LIN {X 70.506,Y 104.962,Z 68.043,A 180.000,B 0.000,C 180.000} C_DIS
LIN {X 70.550,Y 104.810,Z 68.040,A 180.000,B 0.000,C 180.000} C_DIS
LIN {X 70.594,Y 104.659,Z 68.037,A 180.000,B 0.000,C 180.000} C_DIS
LIN {X 70.631,Y 104.506,Z 68.034,A 180.000,B 0.000,C 180.000} C_DIS
LIN {X 70.666,Y 104.352,Z 68.032,A 180.000,B 0.000,C 180.000} C_DIS
LIN {X 70.700,Y 104.199,Z 68.029,A 180.000,B 0.000,C 180.000} C_DIS
LIN {X 70.735,Y 104.045,Z 68.027,A 180.000,B 0.000,C 180.000} C_DIS
LIN {X 70.797,Y 103.736,Z 68.022,A 180.000,B 0.000,C 180.000} C_DIS
LIN {X 70.846,Y 103.425,Z 68.018,A 180.000,B 0.000,C 180.000} C_DIS
LIN {X 70.895,Y 103.114,Z 68.014,A 180.000,B 0.000,C 180.000} C_DIS
LIN {X 70.928,Y 102.801,Z 68.011,A 180.000,B 0.000,C 180.000} C_DIS
LIN {X 70.957,Y 102.487,Z 68.008,A 180.000,B 0.000,C 180.000} C_DIS
LIN {X 70.980,Y 102.173,Z 68.005,A 180.000,B 0.000,C 180.000} C_DIS
LIN {X 70.990,Y 101.858,Z 68.003,A 180.000,B 0.000,C 180.000} C_DIS
LIN {X 71.000,Y 101.543,Z 68.002,A 180.000,B 0.000,C 180.000} C_DIS
LIN {X 70.993,Y 101.228,Z 68.001,A 180.000,B 0.000,C 180.000} C_DIS
LIN {X 70.983,Y 100.914,Z 68.000,A 180.000,B 0.000,C 180.000} C_DIS
LIN {X 70.973,Y 100.682,Z 68.000,A 180.000,B 0.000,C 180.000} C_DIS
; Cutting Move Starts
LIN {X 70.970,Y 100.651,Z 68.000,A 180.000,B 0.000,C 180.000} C_DIS
LIN {X 70.954,Y 100.472,Z 68.000,A 180.000,B 0.000,C 180.000} C_DIS
LIN {X 70.920,Y 100.114,Z 68.000,A 180.000,B 0.000,C 180.000} C_DIS
LIN {X 70.902,Y 99.936,Z 68.000,A 180.000,B 0.000,C 180.000} C_DIS
LIN {X 70.875,Y 99.757,Z 68.000,A 180.000,B 0.000,C 180.000} C_DIS
LIN {X 70.796,Y 99.261,Z 68.000,A 180.000,B 0.000,C 180.000} C_DIS
LIN {X 70.790,Y 99.221,Z 68.000,A 180.000,B 0.000,C 180.000} C_DIS
LIN {X 70.754,Y 99.042,Z 68.000,A 180.000,B 0.000,C 180.000} C_DIS
LIN {X 70.670,Y 98.665,Z 68.000,A 180.000,B 0.000,C 180.000} C_DIS
LIN {X 70.634,Y 98.505,Z 68.000,A 180.000,B 0.000,C 180.000} C_DIS
LIN {X 70.617,Y 98.432,Z 68.000,A 180.000,B 0.000,C 180.000} C_DIS
LIN {X 70.590,Y 98.327,Z 68.000,A 180.000,B 0.000,C 180.000} C_DIS
LIN {X 70.538,Y 98.148,Z 68.000,A 180.000,B 0.000,C 180.000} C_DIS
LIN {X 70.434,Y 97.790,Z 68.000,A 180.000,B 0.000,C 180.000} C_DIS
LIN {X 70.380,Y 97.612,Z 68.000,A 180.000,B 0.000,C 180.000} C_DIS
LIN {X 70.316,Y 97.433,Z 68.000,A 180.000,B 0.000,C 180.000} C_DIS
LIN {X 70.187,Y 97.075,Z 68.000,A 180.000,B 0.000,C 180.000} C_DIS
LIN {X 70.121,Y 96.897,Z 68.000,A 180.000,B 0.000,C 180.000} C_DIS
LIN {X 70.081,Y 96.800,Z 68.000,A 180.000,B 0.000,C 180.000} C_DIS
LIN {X 69.891,Y 96.360,Z 68.000,A 180.000,B 0.000,C 180.000} C_DIS
LIN {X 69.812,Y 96.181,Z 68.000,A 180.000,B 0.000,C 180.000} C_DIS
LIN {X 69.724,Y 96.005,Z 68.000,A 180.000,B 0.000,C 180.000} C_DIS
LIN {X 69.540,Y 95.645,Z 68.000,A 180.000,B 0.000,C 180.000} C_DIS
LIN {X 69.447,Y 95.466,Z 68.000,A 180.000,B 0.000,C 180.000} C_DIS
LIN {X 69.366,Y 95.327,Z 68.000,A 180.000,B 0.000,C 180.000} C_DIS
LIN {X 69.131,Y 94.930,Z 68.000,A 180.000,B 0.000,C 180.000} C_DIS
LIN {X 69.021,Y 94.751,Z 68.000,A 180.000,B 0.000,C 180.000} C_DIS
LIN {X 69.008,Y 94.733,Z 68.000,A 180.000,B 0.000,C 180.000} C_DIS
LIN {X 68.657,Y 94.215,Z 68.000,A 180.000,B 0.000,C 180.000} C_DIS
LIN {X 68.651,Y 94.207,Z 68.000,A 180.000,B 0.000,C 180.000} C_DIS
LIN {X 68.524,Y 94.036,Z 68.000,A 180.000,B 0.000,C 180.000} C_DIS
LIN {X 68.247,Y 93.679,Z 68.000,A 180.000,B 0.000,C 180.000} C_DIS
LIN {X 68.115,Y 93.512,Z 68.000,A 180.000,B 0.000,C 180.000} C_DIS
LIN {X 68.104,Y 93.500,Z 68.000,A 180.000,B 0.000,C 180.000} C_DIS
LIN {X 67.947,Y 93.321,Z 68.000,A 180.000,B 0.000,C 180.000} C_DIS
LIN {X 67.757,Y 93.106,Z 68.000,A 180.000,B 0.000,C 180.000} C_DIS
LIN {X 67.631,Y 92.964,Z 68.000,A 180.000,B 0.000,C 180.000} C_DIS
LIN {X 67.578,Y 92.908,Z 68.000,A 180.000,B 0.000,C 180.000} C_DIS
LIN {X 67.456,Y 92.785,Z 68.000,A 180.000,B 0.000,C 180.000} C_DIS
LIN {X 67.221,Y 92.550,Z 68.000,A 180.000,B 0.000,C 180.000} C_DIS
LIN {X 67.098,Y 92.427,Z 68.000,A 180.000,B 0.000,C 180.000} C_DIS
LIN {X 67.042,Y 92.374,Z 68.000,A 180.000,B 0.000,C 180.000} C_DIS
LIN {X 66.901,Y 92.249,Z 68.000,A 180.000,B 0.000,C 180.000} C_DIS
LIN {X 66.684,Y 92.058,Z 68.000,A 180.000,B 0.000,C 180.000} C_DIS
LIN {X 66.506,Y 91.901,Z 68.000,A 180.000,B 0.000,C 180.000} C_DIS
LIN {X 66.494,Y 91.891,Z 68.000,A 180.000,B 0.000,C 180.000} C_DIS
LIN {X 66.327,Y 91.758,Z 68.000,A 180.000,B 0.000,C 180.000} C_DIS
LIN {X 65.969,Y 91.480,Z 68.000,A 180.000,B 0.000,C 180.000} C_DIS
LIN {X 65.801,Y 91.355,Z 68.000,A 180.000,B 0.000,C 180.000} C_DIS
LIN {X 65.791,Y 91.347,Z 68.000,A 180.000,B 0.000,C 180.000} C_DIS
LIN {X 65.538,Y 91.176,Z 68.000,A 180.000,B 0.000,C 180.000} C_DIS
LIN {X 65.275,Y 90.997,Z 68.000,A 180.000,B 0.000,C 180.000} C_DIS
LIN {X 65.254,Y 90.983,Z 68.000,A 180.000,B 0.000,C 180.000} C_DIS
LIN {X 65.075,Y 90.872,Z 68.000,A 180.000,B 0.000,C 180.000} C_DIS
LIN {X 64.682,Y 90.640,Z 68.000,A 180.000,B 0.000,C 180.000} C_DIS
LIN {X 64.539,Y 90.556,Z 68.000,A 180.000,B 0.000,C 180.000} C_DIS
LIN {X 64.360,Y 90.462,Z 68.000,A 180.000,B 0.000,C 180.000} C_DIS
LIN {X 64.003,Y 90.280,Z 68.000,A 180.000,B 0.000,C 180.000} C_DIS
LIN {X 63.824,Y 90.191,Z 68.000,A 180.000,B 0.000,C 180.000} C_DIS
LIN {X 63.645,Y 90.112,Z 68.000,A 180.000,B 0.000,C 180.000} C_DIS
LIN {X 63.213,Y 89.925,Z 68.000,A 180.000,B 0.000,C 180.000} C_DIS
LIN {X 63.109,Y 89.881,Z 68.000,A 180.000,B 0.000,C 180.000} C_DIS
LIN {X 62.930,Y 89.815,Z 68.000,A 180.000,B 0.000,C 180.000} C_DIS
LIN {X 62.573,Y 89.686,Z 68.000,A 180.000,B 0.000,C 180.000} C_DIS
LIN {X 62.394,Y 89.622,Z 68.000,A 180.000,B 0.000,C 180.000} C_DIS
LIN {X 62.215,Y 89.568,Z 68.000,A 180.000,B 0.000,C 180.000} C_DIS
LIN {X 61.679,Y 89.412,Z 68.000,A 180.000,B 0.000,C 180.000} C_DIS
LIN {X 61.591,Y 89.388,Z 68.000,A 180.000,B 0.000,C 180.000} C_DIS
LIN {X 61.500,Y 89.367,Z 68.000,A 180.000,B 0.000,C 180.000} C_DIS
LIN {X 60.964,Y 89.247,Z 68.000,A 180.000,B 0.000,C 180.000} C_DIS
LIN {X 60.785,Y 89.211,Z 68.000,A 180.000,B 0.000,C 180.000} C_DIS
LIN {X 60.774,Y 89.209,Z 68.000,A 180.000,B 0.000,C 180.000} C_DIS
LIN {X 60.606,Y 89.183,Z 68.000,A 180.000,B 0.000,C 180.000} C_DIS
LIN {X 60.249,Y 89.126,Z 68.000,A 180.000,B 0.000,C 180.000} C_DIS
LIN {X 60.070,Y 89.099,Z 68.000,A 180.000,B 0.000,C 180.000} C_DIS
LIN {X 59.891,Y 89.081,Z 68.000,A 180.000,B 0.000,C 180.000} C_DIS
LIN {X 59.361,Y 89.031,Z 68.000,A 180.000,B 0.000,C 180.000} C_DIS
LIN {X 59.355,Y 89.030,Z 68.000,A 180.000,B 0.000,C 180.000} C_DIS
LIN {X 59.176,Y 89.020,Z 68.000,A 180.000,B 0.000,C 180.000} C_DIS
LIN {X 58.640,Y 89.003,Z 68.000,A 180.000,B 0.000,C 180.000} C_DIS
LIN {X 58.461,Y 89.000,Z 68.000,A 180.000,B 0.000,C 180.000} C_DIS
LIN {X 58.282,Y 89.006,Z 68.000,A 180.000,B 0.000,C 180.000} C_DIS
LIN {X 57.925,Y 89.017,Z 68.000,A 180.000,B 0.000,C 180.000} C_DIS
LIN {X 57.746,Y 89.023,Z 68.000,A 180.000,B 0.000,C 180.000} C_DIS
LIN {X 57.639,Y 89.031,Z 68.000,A 180.000,B 0.000,C 180.000} C_DIS
LIN {X 57.031,Y 89.088,Z 68.000,A 180.000,B 0.000,C 180.000} C_DIS
LIN {X 56.852,Y 89.110,Z 68.000,A 180.000,B 0.000,C 180.000} C_DIS
LIN {X 56.316,Y 89.195,Z 68.000,A 180.000,B 0.000,C 180.000} C_DIS
LIN {X 56.226,Y 89.209,Z 68.000,A 180.000,B 0.000,C 180.000} C_DIS
LIN {X 56.137,Y 89.225,Z 68.000,A 180.000,B 0.000,C 180.000} C_DIS
LIN {X 55.958,Y 89.265,Z 68.000,A 180.000,B 0.000,C 180.000} C_DIS
LIN {X 55.601,Y 89.345,Z 68.000,A 180.000,B 0.000,C 180.000} C_DIS
LIN {X 55.422,Y 89.385,Z 68.000,A 180.000,B 0.000,C 180.000} C_DIS
LIN {X 55.409,Y 89.388,Z 68.000,A 180.000,B 0.000,C 180.000} C_DIS
LIN {X 55.243,Y 89.434,Z 68.000,A 180.000,B 0.000,C 180.000} C_DIS
LIN {X 54.787,Y 89.567,Z 68.000,A 180.000,B 0.000,C 180.000} C_DIS
LIN {X 54.707,Y 89.590,Z 68.000,A 180.000,B 0.000,C 180.000} C_DIS
LIN {X 54.528,Y 89.650,Z 68.000,A 180.000,B 0.000,C 180.000} C_DIS
LIN {X 53.992,Y 89.843,Z 68.000,A 180.000,B 0.000,C 180.000} C_DIS
LIN {X 53.813,Y 89.913,Z 68.000,A 180.000,B 0.000,C 180.000} C_DIS
LIN {X 53.277,Y 90.146,Z 68.000,A 180.000,B 0.000,C 180.000} C_DIS
LIN {X 53.098,Y 90.229,Z 68.000,A 180.000,B 0.000,C 180.000} C_DIS
LIN {X 52.562,Y 90.502,Z 68.000,A 180.000,B 0.000,C 180.000} C_DIS
LIN {X 52.383,Y 90.601,Z 68.000,A 180.000,B 0.000,C 180.000} C_DIS
LIN {X 52.015,Y 90.818,Z 68.000,A 180.000,B 0.000,C 180.000} C_DIS
LIN {X 51.847,Y 90.918,Z 68.000,A 180.000,B 0.000,C 180.000} C_DIS
LIN {X 51.725,Y 90.997,Z 68.000,A 180.000,B 0.000,C 180.000} C_DIS
LIN {X 51.310,Y 91.279,Z 68.000,A 180.000,B 0.000,C 180.000} C_DIS
LIN {X 51.199,Y 91.355,Z 68.000,A 180.000,B 0.000,C 180.000} C_DIS
LIN {X 51.131,Y 91.403,Z 68.000,A 180.000,B 0.000,C 180.000} C_DIS
LIN {X 50.962,Y 91.533,Z 68.000,A 180.000,B 0.000,C 180.000} C_DIS
LIN {X 50.595,Y 91.818,Z 68.000,A 180.000,B 0.000,C 180.000} C_DIS
LIN {X 50.506,Y 91.891,Z 68.000,A 180.000,B 0.000,C 180.000} C_DIS
LIN {X 50.416,Y 91.969,Z 68.000,A 180.000,B 0.000,C 180.000} C_DIS
LIN {X 50.059,Y 92.284,Z 68.000,A 180.000,B 0.000,C 180.000} C_DIS
LIN {X 49.902,Y 92.427,Z 68.000,A 180.000,B 0.000,C 180.000} C_DIS
LIN {X 49.880,Y 92.449,Z 68.000,A 180.000,B 0.000,C 180.000} C_DIS
LIN {X 49.523,Y 92.807,Z 68.000,A 180.000,B 0.000,C 180.000} C_DIS
LIN {X 49.369,Y 92.964,Z 68.000,A 180.000,B 0.000,C 180.000} C_DIS
LIN {X 49.344,Y 92.991,Z 68.000,A 180.000,B 0.000,C 180.000} C_DIS
LIN {X 49.211,Y 93.142,Z 68.000,A 180.000,B 0.000,C 180.000} C_DIS
LIN {X 48.986,Y 93.397,Z 68.000,A 180.000,B 0.000,C 180.000} C_DIS
LIN {X 48.896,Y 93.500,Z 68.000,A 180.000,B 0.000,C 180.000} C_DIS
LIN {X 48.807,Y 93.609,Z 68.000,A 180.000,B 0.000,C 180.000} C_DIS
LIN {X 48.450,Y 94.070,Z 68.000,A 180.000,B 0.000,C 180.000} C_DIS
LIN {X 48.343,Y 94.215,Z 68.000,A 180.000,B 0.000,C 180.000} C_DIS
LIN {X 48.092,Y 94.584,Z 68.000,A 180.000,B 0.000,C 180.000} C_DIS
LIN {X 47.979,Y 94.751,Z 68.000,A 180.000,B 0.000,C 180.000} C_DIS
LIN {X 47.914,Y 94.855,Z 68.000,A 180.000,B 0.000,C 180.000} C_DIS
LIN {X 47.869,Y 94.930,Z 68.000,A 180.000,B 0.000,C 180.000} C_DIS
LIN {X 47.657,Y 95.288,Z 68.000,A 180.000,B 0.000,C 180.000} C_DIS
LIN {X 47.556,Y 95.460,Z 68.000,A 180.000,B 0.000,C 180.000} C_DIS
LIN {X 47.553,Y 95.466,Z 68.000,A 180.000,B 0.000,C 180.000} C_DIS
LIN {X 47.460,Y 95.645,Z 68.000,A 180.000,B 0.000,C 180.000} C_DIS
LIN {X 47.277,Y 96.003,Z 68.000,A 180.000,B 0.000,C 180.000} C_DIS
LIN {X 47.198,Y 96.159,Z 68.000,A 180.000,B 0.000,C 180.000} C_DIS
LIN {X 47.188,Y 96.181,Z 68.000,A 180.000,B 0.000,C 180.000} C_DIS
LIN {X 47.109,Y 96.360,Z 68.000,A 180.000,B 0.000,C 180.000} C_DIS
LIN {X 46.955,Y 96.718,Z 68.000,A 180.000,B 0.000,C 180.000} C_DIS
LIN {X 46.879,Y 96.897,Z 68.000,A 180.000,B 0.000,C 180.000} C_DIS
LIN {X 46.841,Y 96.997,Z 68.000,A 180.000,B 0.000,C 180.000} C_DIS
LIN {X 46.662,Y 97.494,Z 68.000,A 180.000,B 0.000,C 180.000} C_DIS
LIN {X 46.620,Y 97.612,Z 68.000,A 180.000,B 0.000,C 180.000} C_DIS
LIN {X 46.566,Y 97.790,Z 68.000,A 180.000,B 0.000,C 180.000} C_DIS
LIN {X 46.462,Y 98.148,Z 68.000,A 180.000,B 0.000,C 180.000} C_DIS
LIN {X 46.410,Y 98.327,Z 68.000,A 180.000,B 0.000,C 180.000} C_DIS
LIN {X 46.366,Y 98.505,Z 68.000,A 180.000,B 0.000,C 180.000} C_DIS
LIN {X 46.246,Y 99.042,Z 68.000,A 180.000,B 0.000,C 180.000} C_DIS
LIN {X 46.210,Y 99.221,Z 68.000,A 180.000,B 0.000,C 180.000} C_DIS
LIN {X 46.182,Y 99.399,Z 68.000,A 180.000,B 0.000,C 180.000} C_DIS
LIN {X 46.126,Y 99.753,Z 68.000,A 180.000,B 0.000,C 180.000} C_DIS
LIN {X 46.125,Y 99.757,Z 68.000,A 180.000,B 0.000,C 180.000} C_DIS
LIN {X 46.098,Y 99.936,Z 68.000,A 180.000,B 0.000,C 180.000} C_DIS
LIN {X 46.080,Y 100.114,Z 68.000,A 180.000,B 0.000,C 180.000} C_DIS
LIN {X 46.046,Y 100.472,Z 68.000,A 180.000,B 0.000,C 180.000} C_DIS
LIN {X 46.030,Y 100.651,Z 68.000,A 180.000,B 0.000,C 180.000} C_DIS
LIN {X 46.020,Y 100.829,Z 68.000,A 180.000,B 0.000,C 180.000} C_DIS
LIN {X 46.003,Y 101.366,Z 68.000,A 180.000,B 0.000,C 180.000} C_DIS
LIN {X 46.000,Y 101.545,Z 68.000,A 180.000,B 0.000,C 180.000} C_DIS
LIN {X 46.006,Y 101.723,Z 68.000,A 180.000,B 0.000,C 180.000} C_DIS
LIN {X 46.017,Y 102.081,Z 68.000,A 180.000,B 0.000,C 180.000} C_DIS
LIN {X 46.023,Y 102.260,Z 68.000,A 180.000,B 0.000,C 180.000} C_DIS
LIN {X 46.038,Y 102.438,Z 68.000,A 180.000,B 0.000,C 180.000} C_DIS
LIN {X 46.089,Y 102.975,Z 68.000,A 180.000,B 0.000,C 180.000} C_DIS
LIN {X 46.111,Y 103.153,Z 68.000,A 180.000,B 0.000,C 180.000} C_DIS
LIN {X 46.196,Y 103.690,Z 68.000,A 180.000,B 0.000,C 180.000} C_DIS
LIN {X 46.227,Y 103.869,Z 68.000,A 180.000,B 0.000,C 180.000} C_DIS
LIN {X 46.266,Y 104.047,Z 68.000,A 180.000,B 0.000,C 180.000} C_DIS
LIN {X 46.346,Y 104.405,Z 68.000,A 180.000,B 0.000,C 180.000} C_DIS
LIN {X 46.386,Y 104.584,Z 68.000,A 180.000,B 0.000,C 180.000} C_DIS
LIN {X 46.436,Y 104.762,Z 68.000,A 180.000,B 0.000,C 180.000} C_DIS
LIN {X 46.540,Y 105.120,Z 68.000,A 180.000,B 0.000,C 180.000} C_DIS
LIN {X 46.592,Y 105.299,Z 68.000,A 180.000,B 0.000,C 180.000} C_DIS
LIN {X 46.652,Y 105.477,Z 68.000,A 180.000,B 0.000,C 180.000} C_DIS
LIN {X 46.845,Y 106.014,Z 68.000,A 180.000,B 0.000,C 180.000} C_DIS
LIN {X 46.916,Y 106.193,Z 68.000,A 180.000,B 0.000,C 180.000} C_DIS
LIN {X 47.148,Y 106.729,Z 68.000,A 180.000,B 0.000,C 180.000} C_DIS
LIN {X 47.198,Y 106.841,Z 68.000,A 180.000,B 0.000,C 180.000} C_DIS
LIN {X 47.232,Y 106.908,Z 68.000,A 180.000,B 0.000,C 180.000} C_DIS
LIN {X 47.505,Y 107.444,Z 68.000,A 180.000,B 0.000,C 180.000} C_DIS
LIN {X 47.556,Y 107.540,Z 68.000,A 180.000,B 0.000,C 180.000} C_DIS
LIN {X 47.604,Y 107.623,Z 68.000,A 180.000,B 0.000,C 180.000} C_DIS
LIN {X 47.816,Y 107.980,Z 68.000,A 180.000,B 0.000,C 180.000} C_DIS
LIN {X 47.914,Y 108.145,Z 68.000,A 180.000,B 0.000,C 180.000} C_DIS
LIN {X 47.922,Y 108.159,Z 68.000,A 180.000,B 0.000,C 180.000} C_DIS
LIN {X 48.040,Y 108.338,Z 68.000,A 180.000,B 0.000,C 180.000} C_DIS
LIN {X 48.283,Y 108.695,Z 68.000,A 180.000,B 0.000,C 180.000} C_DIS
LIN {X 48.407,Y 108.874,Z 68.000,A 180.000,B 0.000,C 180.000} C_DIS
LIN {X 48.450,Y 108.930,Z 68.000,A 180.000,B 0.000,C 180.000} C_DIS
LIN {X 48.823,Y 109.410,Z 68.000,A 180.000,B 0.000,C 180.000} C_DIS
LIN {X 48.974,Y 109.589,Z 68.000,A 180.000,B 0.000,C 180.000} C_DIS
LIN {X 49.289,Y 109.947,Z 68.000,A 180.000,B 0.000,C 180.000} C_DIS
LIN {X 49.344,Y 110.009,Z 68.000,A 180.000,B 0.000,C 180.000} C_DIS
LIN {X 49.455,Y 110.126,Z 68.000,A 180.000,B 0.000,C 180.000} C_DIS
LIN {X 49.880,Y 110.551,Z 68.000,A 180.000,B 0.000,C 180.000} C_DIS
LIN {X 49.998,Y 110.662,Z 68.000,A 180.000,B 0.000,C 180.000} C_DIS
LIN {X 50.416,Y 111.031,Z 68.000,A 180.000,B 0.000,C 180.000} C_DIS
LIN {X 50.595,Y 111.182,Z 68.000,A 180.000,B 0.000,C 180.000} C_DIS
LIN {X 51.077,Y 111.556,Z 68.000,A 180.000,B 0.000,C 180.000} C_DIS
LIN {X 51.131,Y 111.597,Z 68.000,A 180.000,B 0.000,C 180.000} C_DIS
LIN {X 51.310,Y 111.721,Z 68.000,A 180.000,B 0.000,C 180.000} C_DIS
LIN {X 51.668,Y 111.964,Z 68.000,A 180.000,B 0.000,C 180.000} C_DIS
LIN {X 51.847,Y 112.082,Z 68.000,A 180.000,B 0.000,C 180.000} C_DIS
LIN {X 51.864,Y 112.092,Z 68.000,A 180.000,B 0.000,C 180.000} C_DIS
LIN {X 52.204,Y 112.293,Z 68.000,A 180.000,B 0.000,C 180.000} C_DIS
LIN {X 52.383,Y 112.399,Z 68.000,A 180.000,B 0.000,C 180.000} C_DIS
LIN {X 52.470,Y 112.450,Z 68.000,A 180.000,B 0.000,C 180.000} C_DIS
LIN {X 52.562,Y 112.498,Z 68.000,A 180.000,B 0.000,C 180.000} C_DIS
LIN {X 53.098,Y 112.771,Z 68.000,A 180.000,B 0.000,C 180.000} C_DIS
LIN {X 53.171,Y 112.807,Z 68.000,A 180.000,B 0.000,C 180.000} C_DIS
LIN {X 53.277,Y 112.854,Z 68.000,A 180.000,B 0.000,C 180.000} C_DIS
LIN {X 53.813,Y 113.087,Z 68.000,A 180.000,B 0.000,C 180.000} C_DIS
LIN {X 53.992,Y 113.157,Z 68.000,A 180.000,B 0.000,C 180.000} C_DIS
LIN {X 54.528,Y 113.350,Z 68.000,A 180.000,B 0.000,C 180.000} C_DIS
LIN {X 54.707,Y 113.410,Z 68.000,A 180.000,B 0.000,C 180.000} C_DIS
LIN {X 55.243,Y 113.566,Z 68.000,A 180.000,B 0.000,C 180.000} C_DIS
LIN {X 55.422,Y 113.615,Z 68.000,A 180.000,B 0.000,C 180.000} C_DIS
LIN {X 55.601,Y 113.655,Z 68.000,A 180.000,B 0.000,C 180.000} C_DIS
LIN {X 55.958,Y 113.735,Z 68.000,A 180.000,B 0.000,C 180.000} C_DIS
LIN {X 56.137,Y 113.775,Z 68.000,A 180.000,B 0.000,C 180.000} C_DIS
LIN {X 56.316,Y 113.805,Z 68.000,A 180.000,B 0.000,C 180.000} C_DIS
LIN {X 56.852,Y 113.890,Z 68.000,A 180.000,B 0.000,C 180.000} C_DIS
LIN {X 57.031,Y 113.912,Z 68.000,A 180.000,B 0.000,C 180.000} C_DIS
LIN {X 57.567,Y 113.963,Z 68.000,A 180.000,B 0.000,C 180.000} C_DIS
LIN {X 57.746,Y 113.977,Z 68.000,A 180.000,B 0.000,C 180.000} C_DIS
LIN {X 57.925,Y 113.983,Z 68.000,A 180.000,B 0.000,C 180.000} C_DIS
LIN {X 58.282,Y 113.994,Z 68.000,A 180.000,B 0.000,C 180.000} C_DIS
LIN {X 58.461,Y 114.000,Z 68.000,A 180.000,B 0.000,C 180.000} C_DIS
LIN {X 58.640,Y 113.997,Z 68.000,A 180.000,B 0.000,C 180.000} C_DIS
LIN {X 59.176,Y 113.980,Z 68.000,A 180.000,B 0.000,C 180.000} C_DIS
LIN {X 59.355,Y 113.970,Z 68.000,A 180.000,B 0.000,C 180.000} C_DIS
LIN {X 59.534,Y 113.953,Z 68.000,A 180.000,B 0.000,C 180.000} C_DIS
LIN {X 59.891,Y 113.919,Z 68.000,A 180.000,B 0.000,C 180.000} C_DIS
LIN {X 60.070,Y 113.901,Z 68.000,A 180.000,B 0.000,C 180.000} C_DIS
LIN {X 60.212,Y 113.880,Z 68.000,A 180.000,B 0.000,C 180.000} C_DIS
LIN {X 60.606,Y 113.817,Z 68.000,A 180.000,B 0.000,C 180.000} C_DIS
LIN {X 60.785,Y 113.789,Z 68.000,A 180.000,B 0.000,C 180.000} C_DIS
LIN {X 60.964,Y 113.753,Z 68.000,A 180.000,B 0.000,C 180.000} C_DIS
LIN {X 61.500,Y 113.633,Z 68.000,A 180.000,B 0.000,C 180.000} C_DIS
LIN {X 61.679,Y 113.588,Z 68.000,A 180.000,B 0.000,C 180.000} C_DIS
LIN {X 62.215,Y 113.432,Z 68.000,A 180.000,B 0.000,C 180.000} C_DIS
LIN {X 62.394,Y 113.378,Z 68.000,A 180.000,B 0.000,C 180.000} C_DIS
LIN {X 62.491,Y 113.343,Z 68.000,A 180.000,B 0.000,C 180.000} C_DIS
LIN {X 62.987,Y 113.165,Z 68.000,A 180.000,B 0.000,C 180.000} C_DIS
LIN {X 63.109,Y 113.119,Z 68.000,A 180.000,B 0.000,C 180.000} C_DIS
LIN {X 63.288,Y 113.043,Z 68.000,A 180.000,B 0.000,C 180.000} C_DIS
LIN {X 63.645,Y 112.888,Z 68.000,A 180.000,B 0.000,C 180.000} C_DIS
LIN {X 63.824,Y 112.809,Z 68.000,A 180.000,B 0.000,C 180.000} C_DIS
LIN {X 63.829,Y 112.807,Z 68.000,A 180.000,B 0.000,C 180.000} C_DIS
LIN {X 64.003,Y 112.720,Z 68.000,A 180.000,B 0.000,C 180.000} C_DIS
LIN {X 64.360,Y 112.538,Z 68.000,A 180.000,B 0.000,C 180.000} C_DIS
LIN {X 64.530,Y 112.450,Z 68.000,A 180.000,B 0.000,C 180.000} C_DIS
LIN {X 64.539,Y 112.444,Z 68.000,A 180.000,B 0.000,C 180.000} C_DIS
LIN {X 64.718,Y 112.339,Z 68.000,A 180.000,B 0.000,C 180.000} C_DIS
LIN {X 65.075,Y 112.128,Z 68.000,A 180.000,B 0.000,C 180.000} C_DIS
LIN {X 65.136,Y 112.092,Z 68.000,A 180.000,B 0.000,C 180.000} C_DIS
LIN {X 65.254,Y 112.017,Z 68.000,A 180.000,B 0.000,C 180.000} C_DIS
LIN {X 65.433,Y 111.896,Z 68.000,A 180.000,B 0.000,C 180.000} C_DIS
LIN {X 65.670,Y 111.734,Z 68.000,A 180.000,B 0.000,C 180.000} C_DIS
LIN {X 65.791,Y 111.653,Z 68.000,A 180.000,B 0.000,C 180.000} C_DIS
LIN {X 65.923,Y 111.556,Z 68.000,A 180.000,B 0.000,C 180.000} C_DIS
LIN {X 66.384,Y 111.198,Z 68.000,A 180.000,B 0.000,C 180.000} C_DIS
LIN {X 66.506,Y 111.099,Z 68.000,A 180.000,B 0.000,C 180.000} C_DIS
LIN {X 66.597,Y 111.019,Z 68.000,A 180.000,B 0.000,C 180.000} C_DIS
LIN {X 67.002,Y 110.662,Z 68.000,A 180.000,B 0.000,C 180.000} C_DIS
LIN {X 67.042,Y 110.626,Z 68.000,A 180.000,B 0.000,C 180.000} C_DIS
LIN {X 67.188,Y 110.483,Z 68.000,A 180.000,B 0.000,C 180.000} C_DIS
LIN {X 67.545,Y 110.126,Z 68.000,A 180.000,B 0.000,C 180.000} C_DIS
LIN {X 67.578,Y 110.092,Z 68.000,A 180.000,B 0.000,C 180.000} C_DIS
LIN {X 67.711,Y 109.947,Z 68.000,A 180.000,B 0.000,C 180.000} C_DIS
LIN {X 68.026,Y 109.589,Z 68.000,A 180.000,B 0.000,C 180.000} C_DIS
LIN {X 68.115,Y 109.488,Z 68.000,A 180.000,B 0.000,C 180.000} C_DIS
LIN {X 68.177,Y 109.410,Z 68.000,A 180.000,B 0.000,C 180.000} C_DIS
LIN {X 68.472,Y 109.031,Z 68.000,A 180.000,B 0.000,C 180.000} C_DIS
LIN {X 68.593,Y 108.874,Z 68.000,A 180.000,B 0.000,C 180.000} C_DIS
LIN {X 68.651,Y 108.793,Z 68.000,A 180.000,B 0.000,C 180.000} C_DIS
LIN {X 68.717,Y 108.695,Z 68.000,A 180.000,B 0.000,C 180.000} C_DIS
LIN {X 69.008,Y 108.267,Z 68.000,A 180.000,B 0.000,C 180.000} C_DIS
LIN {X 69.078,Y 108.159,Z 68.000,A 180.000,B 0.000,C 180.000} C_DIS
LIN {X 69.184,Y 107.980,Z 68.000,A 180.000,B 0.000,C 180.000} C_DIS
LIN {X 69.396,Y 107.623,Z 68.000,A 180.000,B 0.000,C 180.000} C_DIS
LIN {X 69.495,Y 107.444,Z 68.000,A 180.000,B 0.000,C 180.000} C_DIS
LIN {X 69.768,Y 106.908,Z 68.000,A 180.000,B 0.000,C 180.000} C_DIS
LIN {X 69.852,Y 106.729,Z 68.000,A 180.000,B 0.000,C 180.000} C_DIS
LIN {X 70.084,Y 106.193,Z 68.000,A 180.000,B 0.000,C 180.000} C_DIS
LIN {X 70.155,Y 106.014,Z 68.000,A 180.000,B 0.000,C 180.000} C_DIS
LIN {X 70.348,Y 105.477,Z 68.000,A 180.000,B 0.000,C 180.000} C_DIS
LIN {X 70.408,Y 105.299,Z 68.000,A 180.000,B 0.000,C 180.000} C_DIS
LIN {X 70.439,Y 105.194,Z 68.000,A 180.000,B 0.000,C 180.000} C_DIS
LIN {X 70.564,Y 104.762,Z 68.000,A 180.000,B 0.000,C 180.000} C_DIS
LIN {X 70.614,Y 104.584,Z 68.000,A 180.000,B 0.000,C 180.000} C_DIS
LIN {X 70.617,Y 104.568,Z 68.000,A 180.000,B 0.000,C 180.000} C_DIS
LIN {X 70.654,Y 104.405,Z 68.000,A 180.000,B 0.000,C 180.000} C_DIS
LIN {X 70.734,Y 104.047,Z 68.000,A 180.000,B 0.000,C 180.000} C_DIS
LIN {X 70.773,Y 103.869,Z 68.000,A 180.000,B 0.000,C 180.000} C_DIS
LIN {X 70.796,Y 103.739,Z 68.000,A 180.000,B 0.000,C 180.000} C_DIS
LIN {X 70.889,Y 103.153,Z 68.000,A 180.000,B 0.000,C 180.000} C_DIS
LIN {X 70.911,Y 102.975,Z 68.000,A 180.000,B 0.000,C 180.000} C_DIS
LIN {X 70.962,Y 102.438,Z 68.000,A 180.000,B 0.000,C 180.000} C_DIS
LIN {X 70.975,Y 102.292,Z 68.000,A 180.000,B 0.000,C 180.000} C_DIS
LIN {X 70.977,Y 102.260,Z 68.000,A 180.000,B 0.000,C 180.000} C_DIS
LIN {X 70.983,Y 102.081,Z 68.000,A 180.000,B 0.000,C 180.000} C_DIS
LIN {X 70.994,Y 101.723,Z 68.000,A 180.000,B 0.000,C 180.000} C_DIS
LIN {X 71.000,Y 101.545,Z 68.000,A 180.000,B 0.000,C 180.000} C_DIS
LIN {X 70.997,Y 101.366,Z 68.000,A 180.000,B 0.000,C 180.000} C_DIS
LIN {X 70.980,Y 100.829,Z 68.000,A 180.000,B 0.000,C 180.000} C_DIS
LIN {X 70.975,Y 100.708,Z 68.000,A 180.000,B 0.000,C 180.000} C_DIS
LIN {X 70.973,Y 100.682,Z 68.000,A 180.000,B 0.000,C 180.000} C_DIS
; Link Move Starts
LIN {X 70.944,Y 100.368,Z 68.000,A 180.000,B 0.000,C 180.000} C_DIS
LIN {X 70.914,Y 100.055,Z 67.999,A 180.000,B 0.000,C 180.000} C_DIS
LIN {X 70.872,Y 99.743,Z 67.998,A 180.000,B 0.000,C 180.000} C_DIS
LIN {X 70.823,Y 99.432,Z 67.996,A 180.000,B 0.000,C 180.000} C_DIS
LIN {X 70.771,Y 99.121,Z 67.994,A 180.000,B 0.000,C 180.000} C_DIS
LIN {X 70.703,Y 98.813,Z 67.991,A 180.000,B 0.000,C 180.000} C_DIS
LIN {X 70.634,Y 98.506,Z 67.988,A 180.000,B 0.000,C 180.000} C_DIS
LIN {X 70.553,Y 98.202,Z 67.985,A 180.000,B 0.000,C 180.000} C_DIS
LIN {X 70.466,Y 97.899,Z 67.981,A 180.000,B 0.000,C 180.000} C_DIS
LIN {X 70.375,Y 97.597,Z 67.977,A 180.000,B 0.000,C 180.000} C_DIS
LIN {X 70.268,Y 97.301,Z 67.972,A 180.000,B 0.000,C 180.000} C_DIS
LIN {X 70.215,Y 97.153,Z 67.969,A 180.000,B 0.000,C 180.000} C_DIS
LIN {X 70.162,Y 97.005,Z 67.967,A 180.000,B 0.000,C 180.000} C_DIS
LIN {X 70.106,Y 96.857,Z 67.964,A 180.000,B 0.000,C 180.000} C_DIS
LIN {X 70.043,Y 96.713,Z 67.961,A 180.000,B 0.000,C 180.000} C_DIS
LIN {X 69.981,Y 96.568,Z 67.959,A 180.000,B 0.000,C 180.000} C_DIS
LIN {X 69.918,Y 96.424,Z 67.956,A 180.000,B 0.000,C 180.000} C_DIS
LIN {X 69.856,Y 96.279,Z 67.952,A 180.000,B 0.000,C 180.000} C_DIS
LIN {X 69.790,Y 96.136,Z 67.949,A 180.000,B 0.000,C 180.000} C_DIS
LIN {X 69.719,Y 95.995,Z 67.946,A 180.000,B 0.000,C 180.000} C_DIS
LIN {X 69.647,Y 95.855,Z 67.943,A 180.000,B 0.000,C 180.000} C_DIS
LIN {X 69.576,Y 95.715,Z 67.939,A 180.000,B 0.000,C 180.000} C_DIS
LIN {X 69.504,Y 95.574,Z 67.936,A 180.000,B 0.000,C 180.000} C_DIS
LIN {X 69.430,Y 95.436,Z 67.932,A 180.000,B 0.000,C 180.000} C_DIS
LIN {X 69.350,Y 95.300,Z 67.928,A 180.000,B 0.000,C 180.000} C_DIS
LIN {X 69.270,Y 95.164,Z 67.925,A 180.000,B 0.000,C 180.000} C_DIS
LIN {X 69.190,Y 95.029,Z 67.921,A 180.000,B 0.000,C 180.000} C_DIS
LIN {X 69.109,Y 94.893,Z 67.917,A 180.000,B 0.000,C 180.000} C_DIS
LIN {X 69.026,Y 94.759,Z 67.913,A 180.000,B 0.000,C 180.000} C_DIS
LIN {X 68.938,Y 94.629,Z 67.909,A 180.000,B 0.000,C 180.000} C_DIS
LIN {X 68.849,Y 94.499,Z 67.905,A 180.000,B 0.000,C 180.000} C_DIS
LIN {X 68.761,Y 94.369,Z 67.900,A 180.000,B 0.000,C 180.000} C_DIS
LIN {X 68.672,Y 94.238,Z 67.896,A 180.000,B 0.000,C 180.000} C_DIS
LIN {X 68.581,Y 94.110,Z 67.892,A 180.000,B 0.000,C 180.000} C_DIS
LIN {X 68.485,Y 93.985,Z 67.887,A 180.000,B 0.000,C 180.000} C_DIS
LIN {X 68.388,Y 93.861,Z 67.883,A 180.000,B 0.000,C 180.000} C_DIS
LIN {X 68.292,Y 93.737,Z 67.878,A 180.000,B 0.000,C 180.000} C_DIS
LIN {X 68.195,Y 93.612,Z 67.873,A 180.000,B 0.000,C 180.000} C_DIS
LIN {X 68.096,Y 93.490,Z 67.869,A 180.000,B 0.000,C 180.000} C_DIS
LIN {X 67.992,Y 93.372,Z 67.864,A 180.000,B 0.000,C 180.000} C_DIS
LIN {X 67.887,Y 93.254,Z 67.859,A 180.000,B 0.000,C 180.000} C_DIS
LIN {X 67.783,Y 93.135,Z 67.854,A 180.000,B 0.000,C 180.000} C_DIS
LIN {X 67.731,Y 93.076,Z 67.851,A 180.000,B 0.000,C 180.000} C_DIS
LIN {X 67.679,Y 93.017,Z 67.849,A 180.000,B 0.000,C 180.000} C_DIS
LIN {X 67.627,Y 92.959,Z 67.846,A 180.000,B 0.000,C 180.000} C_DIS
LIN {X 67.572,Y 92.902,Z 67.844,A 180.000,B 0.000,C 180.000} C_DIS
LIN {X 67.517,Y 92.846,Z 67.841,A 180.000,B 0.000,C 180.000} C_DIS
LIN {X 67.461,Y 92.790,Z 67.839,A 180.000,B 0.000,C 180.000} C_DIS
LIN {X 67.405,Y 92.735,Z 67.836,A 180.000,B 0.000,C 180.000} C_DIS
LIN {X 67.294,Y 92.623,Z 67.831,A 180.000,B 0.000,C 180.000} C_DIS
LIN {X 67.182,Y 92.512,Z 67.825,A 180.000,B 0.000,C 180.000} C_DIS
LIN {X 67.127,Y 92.456,Z 67.823,A 180.000,B 0.000,C 180.000} C_DIS
LIN {X 67.071,Y 92.401,Z 67.820,A 180.000,B 0.000,C 180.000} C_DIS
LIN {X 67.013,Y 92.347,Z 67.817,A 180.000,B 0.000,C 180.000} C_DIS
LIN {X 66.954,Y 92.295,Z 67.815,A 180.000,B 0.000,C 180.000} C_DIS
LIN {X 66.836,Y 92.191,Z 67.809,A 180.000,B 0.000,C 180.000} C_DIS
LIN {X 66.777,Y 92.139,Z 67.807,A 180.000,B 0.000,C 180.000} C_DIS
LIN {X 66.658,Y 92.035,Z 67.801,A 180.000,B 0.000,C 180.000} C_DIS
LIN {X 66.540,Y 91.931,Z 67.796,A 180.000,B 0.000,C 180.000} C_DIS
LIN {X 66.481,Y 91.879,Z 67.793,A 180.000,B 0.000,C 180.000} C_DIS
LIN {X 66.420,Y 91.830,Z 67.790,A 180.000,B 0.000,C 180.000} C_DIS
LIN {X 66.357,Y 91.781,Z 67.787,A 180.000,B 0.000,C 180.000} C_DIS
LIN {X 66.295,Y 91.733,Z 67.785,A 180.000,B 0.000,C 180.000} C_DIS
LIN {X 66.171,Y 91.637,Z 67.779,A 180.000,B 0.000,C 180.000} C_DIS
LIN {X 65.984,Y 91.492,Z 67.771,A 180.000,B 0.000,C 180.000} C_DIS
LIN {X 65.922,Y 91.443,Z 67.768,A 180.000,B 0.000,C 180.000} C_DIS
LIN {X 65.859,Y 91.396,Z 67.765,A 180.000,B 0.000,C 180.000} C_DIS
LIN {X 65.795,Y 91.350,Z 67.763,A 180.000,B 0.000,C 180.000} C_DIS
LIN {X 65.730,Y 91.306,Z 67.760,A 180.000,B 0.000,C 180.000} C_DIS
LIN {X 65.599,Y 91.217,Z 67.754,A 180.000,B 0.000,C 180.000} C_DIS
LIN {X 65.534,Y 91.173,Z 67.752,A 180.000,B 0.000,C 180.000} C_DIS
LIN {X 65.404,Y 91.085,Z 67.746,A 180.000,B 0.000,C 180.000} C_DIS
LIN {X 65.274,Y 90.996,Z 67.741,A 180.000,B 0.000,C 180.000} C_DIS
LIN {X 65.208,Y 90.953,Z 67.738,A 180.000,B 0.000,C 180.000} C_DIS
LIN {X 65.141,Y 90.911,Z 67.735,A 180.000,B 0.000,C 180.000} C_DIS
LIN {X 65.073,Y 90.871,Z 67.732,A 180.000,B 0.000,C 180.000} C_DIS
LIN {X 65.006,Y 90.831,Z 67.730,A 180.000,B 0.000,C 180.000} C_DIS
LIN {X 64.870,Y 90.751,Z 67.724,A 180.000,B 0.000,C 180.000} C_DIS
LIN {X 64.599,Y 90.590,Z 67.713,A 180.000,B 0.000,C 180.000} C_DIS
LIN {X 64.531,Y 90.551,Z 67.710,A 180.000,B 0.000,C 180.000} C_DIS
LIN {X 64.461,Y 90.514,Z 67.708,A 180.000,B 0.000,C 180.000} C_DIS
LIN {X 64.391,Y 90.478,Z 67.705,A 180.000,B 0.000,C 180.000} C_DIS
LIN {X 64.251,Y 90.407,Z 67.699,A 180.000,B 0.000,C 180.000} C_DIS
LIN {X 64.181,Y 90.371,Z 67.697,A 180.000,B 0.000,C 180.000} C_DIS
LIN {X 64.040,Y 90.299,Z 67.691,A 180.000,B 0.000,C 180.000} C_DIS
LIN {X 63.900,Y 90.228,Z 67.686,A 180.000,B 0.000,C 180.000} C_DIS
LIN {X 63.829,Y 90.193,Z 67.683,A 180.000,B 0.000,C 180.000} C_DIS
LIN {X 63.758,Y 90.160,Z 67.680,A 180.000,B 0.000,C 180.000} C_DIS
LIN {X 63.613,Y 90.098,Z 67.675,A 180.000,B 0.000,C 180.000} C_DIS
LIN {X 63.469,Y 90.035,Z 67.669,A 180.000,B 0.000,C 180.000} C_DIS
LIN {X 63.179,Y 89.910,Z 67.658,A 180.000,B 0.000,C 180.000} C_DIS
LIN {X 63.107,Y 89.880,Z 67.655,A 180.000,B 0.000,C 180.000} C_DIS
LIN {X 63.033,Y 89.852,Z 67.653,A 180.000,B 0.000,C 180.000} C_DIS
LIN {X 62.885,Y 89.799,Z 67.647,A 180.000,B 0.000,C 180.000} C_DIS
LIN {X 62.440,Y 89.638,Z 67.631,A 180.000,B 0.000,C 180.000} C_DIS
LIN {X 62.366,Y 89.613,Z 67.628,A 180.000,B 0.000,C 180.000} C_DIS
LIN {X 62.291,Y 89.590,Z 67.625,A 180.000,B 0.000,C 180.000} C_DIS
LIN {X 61.761,Y 89.436,Z 67.606,A 180.000,B 0.000,C 180.000} C_DIS
LIN {X 61.686,Y 89.414,Z 67.603,A 180.000,B 0.000,C 180.000} C_DIS
LIN {X 61.610,Y 89.393,Z 67.600,A 180.000,B 0.000,C 180.000} C_DIS
LIN {X 61.533,Y 89.375,Z 67.598,A 180.000,B 0.000,C 180.000} C_DIS
LIN {X 61.303,Y 89.323,Z 67.589,A 180.000,B 0.000,C 180.000} C_DIS
LIN {X 60.995,Y 89.254,Z 67.578,A 180.000,B 0.000,C 180.000} C_DIS
LIN {X 60.918,Y 89.237,Z 67.576,A 180.000,B 0.000,C 180.000} C_DIS
LIN {X 60.841,Y 89.221,Z 67.573,A 180.000,B 0.000,C 180.000} C_DIS
LIN {X 60.764,Y 89.208,Z 67.570,A 180.000,B 0.000,C 180.000} C_DIS
LIN {X 60.141,Y 89.109,Z 67.548,A 180.000,B 0.000,C 180.000} C_DIS
LIN {X 60.063,Y 89.098,Z 67.545,A 180.000,B 0.000,C 180.000} C_DIS
LIN {X 59.985,Y 89.090,Z 67.543,A 180.000,B 0.000,C 180.000} C_DIS
LIN {X 59.358,Y 89.030,Z 67.521,A 180.000,B 0.000,C 180.000} C_DIS
LIN {X 59.279,Y 89.024,Z 67.518,A 180.000,B 0.000,C 180.000} C_DIS
LIN {X 59.201,Y 89.021,Z 67.515,A 180.000,B 0.000,C 180.000} C_DIS
LIN {X 58.571,Y 89.001,Z 67.493,A 180.000,B 0.000,C 180.000} C_DIS
LIN {X 58.492,Y 89.000,Z 67.490,A 180.000,B 0.000,C 180.000} C_DIS
LIN {X 58.414,Y 89.001,Z 67.488,A 180.000,B 0.000,C 180.000} C_DIS
LIN {X 57.863,Y 89.019,Z 67.468,A 180.000,B 0.000,C 180.000} C_DIS
LIN {X 57.784,Y 89.021,Z 67.466,A 180.000,B 0.000,C 180.000} C_DIS
LIN {X 57.705,Y 89.025,Z 67.463,A 180.000,B 0.000,C 180.000} C_DIS
LIN {X 57.627,Y 89.032,Z 67.460,A 180.000,B 0.000,C 180.000} C_DIS
LIN {X 57.078,Y 89.084,Z 67.441,A 180.000,B 0.000,C 180.000} C_DIS
LIN {X 56.999,Y 89.091,Z 67.438,A 180.000,B 0.000,C 180.000} C_DIS
LIN {X 56.921,Y 89.100,Z 67.435,A 180.000,B 0.000,C 180.000} C_DIS
LIN {X 56.843,Y 89.112,Z 67.433,A 180.000,B 0.000,C 180.000} C_DIS
LIN {X 56.377,Y 89.185,Z 67.416,A 180.000,B 0.000,C 180.000} C_DIS
LIN {X 56.299,Y 89.198,Z 67.413,A 180.000,B 0.000,C 180.000} C_DIS
LIN {X 56.221,Y 89.210,Z 67.411,A 180.000,B 0.000,C 180.000} C_DIS
LIN {X 56.144,Y 89.224,Z 67.408,A 180.000,B 0.000,C 180.000} C_DIS
LIN {X 56.067,Y 89.241,Z 67.405,A 180.000,B 0.000,C 180.000} C_DIS
LIN {X 55.529,Y 89.361,Z 67.386,A 180.000,B 0.000,C 180.000} C_DIS
LIN {X 55.452,Y 89.378,Z 67.383,A 180.000,B 0.000,C 180.000} C_DIS
LIN {X 55.375,Y 89.397,Z 67.380,A 180.000,B 0.000,C 180.000} C_DIS
LIN {X 55.299,Y 89.418,Z 67.378,A 180.000,B 0.000,C 180.000} C_DIS
LIN {X 55.073,Y 89.484,Z 67.369,A 180.000,B 0.000,C 180.000} C_DIS
LIN {X 54.921,Y 89.528,Z 67.364,A 180.000,B 0.000,C 180.000} C_DIS
LIN {X 54.770,Y 89.572,Z 67.358,A 180.000,B 0.000,C 180.000} C_DIS
LIN {X 54.694,Y 89.594,Z 67.356,A 180.000,B 0.000,C 180.000} C_DIS
LIN {X 54.619,Y 89.618,Z 67.353,A 180.000,B 0.000,C 180.000} C_DIS
LIN {X 54.545,Y 89.644,Z 67.350,A 180.000,B 0.000,C 180.000} C_DIS
LIN {X 54.026,Y 89.830,Z 67.331,A 180.000,B 0.000,C 180.000} C_DIS
LIN {X 53.952,Y 89.857,Z 67.328,A 180.000,B 0.000,C 180.000} C_DIS
LIN {X 53.879,Y 89.886,Z 67.325,A 180.000,B 0.000,C 180.000} C_DIS
LIN {X 53.806,Y 89.916,Z 67.323,A 180.000,B 0.000,C 180.000} C_DIS
LIN {X 53.662,Y 89.979,Z 67.317,A 180.000,B 0.000,C 180.000} C_DIS
LIN {X 53.300,Y 90.135,Z 67.303,A 180.000,B 0.000,C 180.000} C_DIS
LIN {X 53.228,Y 90.167,Z 67.301,A 180.000,B 0.000,C 180.000} C_DIS
LIN {X 53.157,Y 90.200,Z 67.298,A 180.000,B 0.000,C 180.000} C_DIS
LIN {X 53.086,Y 90.235,Z 67.295,A 180.000,B 0.000,C 180.000} C_DIS
LIN {X 52.665,Y 90.449,Z 67.279,A 180.000,B 0.000,C 180.000} C_DIS
LIN {X 52.595,Y 90.485,Z 67.276,A 180.000,B 0.000,C 180.000} C_DIS
LIN {X 52.525,Y 90.521,Z 67.273,A 180.000,B 0.000,C 180.000} C_DIS
LIN {X 52.456,Y 90.559,Z 67.270,A 180.000,B 0.000,C 180.000} C_DIS
LIN {X 52.388,Y 90.598,Z 67.268,A 180.000,B 0.000,C 180.000} C_DIS
LIN {X 52.252,Y 90.678,Z 67.262,A 180.000,B 0.000,C 180.000} C_DIS
LIN {X 52.049,Y 90.799,Z 67.254,A 180.000,B 0.000,C 180.000} C_DIS
LIN {X 51.913,Y 90.879,Z 67.248,A 180.000,B 0.000,C 180.000} C_DIS
LIN {X 51.845,Y 90.919,Z 67.246,A 180.000,B 0.000,C 180.000} C_DIS
LIN {X 51.779,Y 90.961,Z 67.243,A 180.000,B 0.000,C 180.000} C_DIS
LIN {X 51.713,Y 91.005,Z 67.240,A 180.000,B 0.000,C 180.000} C_DIS
LIN {X 51.518,Y 91.138,Z 67.232,A 180.000,B 0.000,C 180.000} C_DIS
LIN {X 51.388,Y 91.226,Z 67.226,A 180.000,B 0.000,C 180.000} C_DIS
LIN {X 51.323,Y 91.270,Z 67.224,A 180.000,B 0.000,C 180.000} C_DIS
LIN {X 51.257,Y 91.315,Z 67.221,A 180.000,B 0.000,C 180.000} C_DIS
LIN {X 51.192,Y 91.359,Z 67.218,A 180.000,B 0.000,C 180.000} C_DIS
LIN {X 51.128,Y 91.405,Z 67.215,A 180.000,B 0.000,C 180.000} C_DIS
LIN {X 51.066,Y 91.453,Z 67.213,A 180.000,B 0.000,C 180.000} C_DIS
LIN {X 50.942,Y 91.550,Z 67.207,A 180.000,B 0.000,C 180.000} C_DIS
LIN {X 50.755,Y 91.694,Z 67.199,A 180.000,B 0.000,C 180.000} C_DIS
LIN {X 50.630,Y 91.791,Z 67.193,A 180.000,B 0.000,C 180.000} C_DIS
LIN {X 50.568,Y 91.839,Z 67.191,A 180.000,B 0.000,C 180.000} C_DIS
LIN {X 50.507,Y 91.889,Z 67.188,A 180.000,B 0.000,C 180.000} C_DIS
LIN {X 50.448,Y 91.941,Z 67.185,A 180.000,B 0.000,C 180.000} C_DIS
LIN {X 50.330,Y 92.045,Z 67.180,A 180.000,B 0.000,C 180.000} C_DIS
LIN {X 50.212,Y 92.149,Z 67.174,A 180.000,B 0.000,C 180.000} C_DIS
LIN {X 50.094,Y 92.254,Z 67.169,A 180.000,B 0.000,C 180.000} C_DIS
LIN {X 50.035,Y 92.306,Z 67.166,A 180.000,B 0.000,C 180.000} C_DIS
LIN {X 49.976,Y 92.358,Z 67.164,A 180.000,B 0.000,C 180.000} C_DIS
LIN {X 49.918,Y 92.412,Z 67.161,A 180.000,B 0.000,C 180.000} C_DIS
LIN {X 49.862,Y 92.467,Z 67.159,A 180.000,B 0.000,C 180.000} C_DIS
LIN {X 49.807,Y 92.523,Z 67.156,A 180.000,B 0.000,C 180.000} C_DIS
LIN {X 49.751,Y 92.578,Z 67.154,A 180.000,B 0.000,C 180.000} C_DIS
LIN {X 49.695,Y 92.634,Z 67.151,A 180.000,B 0.000,C 180.000} C_DIS
LIN {X 49.639,Y 92.690,Z 67.149,A 180.000,B 0.000,C 180.000} C_DIS
LIN {X 49.528,Y 92.801,Z 67.144,A 180.000,B 0.000,C 180.000} C_DIS
LIN {X 49.417,Y 92.913,Z 67.139,A 180.000,B 0.000,C 180.000} C_DIS
LIN {X 49.311,Y 93.029,Z 67.134,A 180.000,B 0.000,C 180.000} C_DIS
LIN {X 49.206,Y 93.147,Z 67.129,A 180.000,B 0.000,C 180.000} C_DIS
LIN {X 49.102,Y 93.265,Z 67.124,A 180.000,B 0.000,C 180.000} C_DIS
LIN {X 48.998,Y 93.383,Z 67.120,A 180.000,B 0.000,C 180.000} C_DIS
LIN {X 48.894,Y 93.502,Z 67.115,A 180.000,B 0.000,C 180.000} C_DIS
LIN {X 48.795,Y 93.624,Z 67.111,A 180.000,B 0.000,C 180.000} C_DIS
LIN {X 48.699,Y 93.749,Z 67.106,A 180.000,B 0.000,C 180.000} C_DIS
LIN {X 48.602,Y 93.873,Z 67.102,A 180.000,B 0.000,C 180.000} C_DIS
LIN {X 48.506,Y 93.998,Z 67.097,A 180.000,B 0.000,C 180.000} C_DIS
LIN {X 48.410,Y 94.122,Z 67.093,A 180.000,B 0.000,C 180.000} C_DIS
LIN {X 48.319,Y 94.251,Z 67.089,A 180.000,B 0.000,C 180.000} C_DIS
LIN {X 48.230,Y 94.381,Z 67.085,A 180.000,B 0.000,C 180.000} C_DIS
LIN {X 48.142,Y 94.512,Z 67.081,A 180.000,B 0.000,C 180.000} C_DIS
LIN {X 48.053,Y 94.642,Z 67.077,A 180.000,B 0.000,C 180.000} C_DIS
LIN {X 47.965,Y 94.772,Z 67.073,A 180.000,B 0.000,C 180.000} C_DIS
LIN {X 47.883,Y 94.907,Z 67.070,A 180.000,B 0.000,C 180.000} C_DIS
LIN {X 47.802,Y 95.042,Z 67.066,A 180.000,B 0.000,C 180.000} C_DIS
LIN {X 47.722,Y 95.178,Z 67.062,A 180.000,B 0.000,C 180.000} C_DIS
LIN {X 47.642,Y 95.313,Z 67.059,A 180.000,B 0.000,C 180.000} C_DIS
LIN {X 47.562,Y 95.449,Z 67.056,A 180.000,B 0.000,C 180.000} C_DIS
LIN {X 47.489,Y 95.588,Z 67.052,A 180.000,B 0.000,C 180.000} C_DIS
LIN {X 47.417,Y 95.729,Z 67.049,A 180.000,B 0.000,C 180.000} C_DIS
LIN {X 47.346,Y 95.869,Z 67.046,A 180.000,B 0.000,C 180.000} C_DIS
LIN {X 47.274,Y 96.009,Z 67.043,A 180.000,B 0.000,C 180.000} C_DIS
LIN {X 47.203,Y 96.150,Z 67.040,A 180.000,B 0.000,C 180.000} C_DIS
LIN {X 47.138,Y 96.293,Z 67.037,A 180.000,B 0.000,C 180.000} C_DIS
LIN {X 47.076,Y 96.438,Z 67.034,A 180.000,B 0.000,C 180.000} C_DIS
LIN {X 47.013,Y 96.583,Z 67.032,A 180.000,B 0.000,C 180.000} C_DIS
LIN {X 46.951,Y 96.727,Z 67.029,A 180.000,B 0.000,C 180.000} C_DIS
LIN {X 46.889,Y 96.872,Z 67.027,A 180.000,B 0.000,C 180.000} C_DIS
LIN {X 46.780,Y 97.167,Z 67.022,A 180.000,B 0.000,C 180.000} C_DIS
LIN {X 46.673,Y 97.464,Z 67.018,A 180.000,B 0.000,C 180.000} C_DIS
LIN {X 46.574,Y 97.763,Z 67.014,A 180.000,B 0.000,C 180.000} C_DIS
LIN {X 46.486,Y 98.065,Z 67.011,A 180.000,B 0.000,C 180.000} C_DIS
LIN {X 46.399,Y 98.368,Z 67.008,A 180.000,B 0.000,C 180.000} C_DIS
LIN {X 46.328,Y 98.675,Z 67.005,A 180.000,B 0.000,C 180.000} C_DIS
LIN {X 46.259,Y 98.982,Z 67.003,A 180.000,B 0.000,C 180.000} C_DIS
LIN {X 46.199,Y 99.291,Z 67.002,A 180.000,B 0.000,C 180.000} C_DIS
LIN {X 46.150,Y 99.602,Z 67.001,A 180.000,B 0.000,C 180.000} C_DIS
LIN {X 46.101,Y 99.914,Z 67.000,A 180.000,B 0.000,C 180.000} C_DIS
LIN {X 46.077,Y 100.144,Z 67.000,A 180.000,B 0.000,C 180.000} C_DIS
; Cutting Move Starts
LIN {X 46.046,Y 100.472,Z 67.000,A 180.000,B 0.000,C 180.000} C_DIS
LIN {X 46.030,Y 100.651,Z 67.000,A 180.000,B 0.000,C 180.000} C_DIS
LIN {X 46.020,Y 100.829,Z 67.000,A 180.000,B 0.000,C 180.000} C_DIS
LIN {X 46.003,Y 101.366,Z 67.000,A 180.000,B 0.000,C 180.000} C_DIS
LIN {X 46.000,Y 101.545,Z 67.000,A 180.000,B 0.000,C 180.000} C_DIS
LIN {X 46.006,Y 101.723,Z 67.000,A 180.000,B 0.000,C 180.000} C_DIS
LIN {X 46.017,Y 102.081,Z 67.000,A 180.000,B 0.000,C 180.000} C_DIS
LIN {X 46.023,Y 102.260,Z 67.000,A 180.000,B 0.000,C 180.000} C_DIS
LIN {X 46.038,Y 102.438,Z 67.000,A 180.000,B 0.000,C 180.000} C_DIS
LIN {X 46.089,Y 102.975,Z 67.000,A 180.000,B 0.000,C 180.000} C_DIS
LIN {X 46.111,Y 103.153,Z 67.000,A 180.000,B 0.000,C 180.000} C_DIS
LIN {X 46.196,Y 103.690,Z 67.000,A 180.000,B 0.000,C 180.000} C_DIS
LIN {X 46.227,Y 103.869,Z 67.000,A 180.000,B 0.000,C 180.000} C_DIS
LIN {X 46.266,Y 104.047,Z 67.000,A 180.000,B 0.000,C 180.000} C_DIS
LIN {X 46.346,Y 104.405,Z 67.000,A 180.000,B 0.000,C 180.000} C_DIS
LIN {X 46.386,Y 104.584,Z 67.000,A 180.000,B 0.000,C 180.000} C_DIS
LIN {X 46.436,Y 104.762,Z 67.000,A 180.000,B 0.000,C 180.000} C_DIS
LIN {X 46.540,Y 105.120,Z 67.000,A 180.000,B 0.000,C 180.000} C_DIS
LIN {X 46.592,Y 105.299,Z 67.000,A 180.000,B 0.000,C 180.000} C_DIS
LIN {X 46.652,Y 105.477,Z 67.000,A 180.000,B 0.000,C 180.000} C_DIS
LIN {X 46.845,Y 106.014,Z 67.000,A 180.000,B 0.000,C 180.000} C_DIS
LIN {X 46.916,Y 106.193,Z 67.000,A 180.000,B 0.000,C 180.000} C_DIS
LIN {X 47.148,Y 106.729,Z 67.000,A 180.000,B 0.000,C 180.000} C_DIS
LIN {X 47.198,Y 106.841,Z 67.000,A 180.000,B 0.000,C 180.000} C_DIS
LIN {X 47.232,Y 106.908,Z 67.000,A 180.000,B 0.000,C 180.000} C_DIS
LIN {X 47.505,Y 107.444,Z 67.000,A 180.000,B 0.000,C 180.000} C_DIS
LIN {X 47.556,Y 107.540,Z 67.000,A 180.000,B 0.000,C 180.000} C_DIS
LIN {X 47.604,Y 107.623,Z 67.000,A 180.000,B 0.000,C 180.000} C_DIS
LIN {X 47.816,Y 107.980,Z 67.000,A 180.000,B 0.000,C 180.000} C_DIS
LIN {X 47.914,Y 108.145,Z 67.000,A 180.000,B 0.000,C 180.000} C_DIS
LIN {X 47.922,Y 108.159,Z 67.000,A 180.000,B 0.000,C 180.000} C_DIS
LIN {X 48.040,Y 108.338,Z 67.000,A 180.000,B 0.000,C 180.000} C_DIS
LIN {X 48.283,Y 108.695,Z 67.000,A 180.000,B 0.000,C 180.000} C_DIS
LIN {X 48.407,Y 108.874,Z 67.000,A 180.000,B 0.000,C 180.000} C_DIS
LIN {X 48.450,Y 108.930,Z 67.000,A 180.000,B 0.000,C 180.000} C_DIS
LIN {X 48.823,Y 109.410,Z 67.000,A 180.000,B 0.000,C 180.000} C_DIS
LIN {X 48.974,Y 109.589,Z 67.000,A 180.000,B 0.000,C 180.000} C_DIS
LIN {X 49.289,Y 109.947,Z 67.000,A 180.000,B 0.000,C 180.000} C_DIS
LIN {X 49.344,Y 110.009,Z 67.000,A 180.000,B 0.000,C 180.000} C_DIS
LIN {X 49.455,Y 110.126,Z 67.000,A 180.000,B 0.000,C 180.000} C_DIS
LIN {X 49.880,Y 110.551,Z 67.000,A 180.000,B 0.000,C 180.000} C_DIS
LIN {X 49.998,Y 110.662,Z 67.000,A 180.000,B 0.000,C 180.000} C_DIS
LIN {X 50.416,Y 111.031,Z 67.000,A 180.000,B 0.000,C 180.000} C_DIS
LIN {X 50.595,Y 111.182,Z 67.000,A 180.000,B 0.000,C 180.000} C_DIS
LIN {X 51.077,Y 111.556,Z 67.000,A 180.000,B 0.000,C 180.000} C_DIS
LIN {X 51.131,Y 111.597,Z 67.000,A 180.000,B 0.000,C 180.000} C_DIS
LIN {X 51.310,Y 111.721,Z 67.000,A 180.000,B 0.000,C 180.000} C_DIS
LIN {X 51.668,Y 111.964,Z 67.000,A 180.000,B 0.000,C 180.000} C_DIS
LIN {X 51.847,Y 112.082,Z 67.000,A 180.000,B 0.000,C 180.000} C_DIS
LIN {X 51.864,Y 112.092,Z 67.000,A 180.000,B 0.000,C 180.000} C_DIS
LIN {X 52.204,Y 112.293,Z 67.000,A 180.000,B 0.000,C 180.000} C_DIS
LIN {X 52.383,Y 112.399,Z 67.000,A 180.000,B 0.000,C 180.000} C_DIS
LIN {X 52.470,Y 112.450,Z 67.000,A 180.000,B 0.000,C 180.000} C_DIS
LIN {X 52.562,Y 112.498,Z 67.000,A 180.000,B 0.000,C 180.000} C_DIS
LIN {X 53.098,Y 112.771,Z 67.000,A 180.000,B 0.000,C 180.000} C_DIS
LIN {X 53.171,Y 112.807,Z 67.000,A 180.000,B 0.000,C 180.000} C_DIS
LIN {X 53.277,Y 112.854,Z 67.000,A 180.000,B 0.000,C 180.000} C_DIS
LIN {X 53.813,Y 113.087,Z 67.000,A 180.000,B 0.000,C 180.000} C_DIS
LIN {X 53.992,Y 113.157,Z 67.000,A 180.000,B 0.000,C 180.000} C_DIS
LIN {X 54.528,Y 113.350,Z 67.000,A 180.000,B 0.000,C 180.000} C_DIS
LIN {X 54.707,Y 113.410,Z 67.000,A 180.000,B 0.000,C 180.000} C_DIS
LIN {X 55.243,Y 113.566,Z 67.000,A 180.000,B 0.000,C 180.000} C_DIS
LIN {X 55.422,Y 113.615,Z 67.000,A 180.000,B 0.000,C 180.000} C_DIS
LIN {X 55.601,Y 113.655,Z 67.000,A 180.000,B 0.000,C 180.000} C_DIS
LIN {X 55.958,Y 113.735,Z 67.000,A 180.000,B 0.000,C 180.000} C_DIS
LIN {X 56.137,Y 113.775,Z 67.000,A 180.000,B 0.000,C 180.000} C_DIS
LIN {X 56.316,Y 113.805,Z 67.000,A 180.000,B 0.000,C 180.000} C_DIS
LIN {X 56.852,Y 113.890,Z 67.000,A 180.000,B 0.000,C 180.000} C_DIS
LIN {X 57.031,Y 113.912,Z 67.000,A 180.000,B 0.000,C 180.000} C_DIS
LIN {X 57.567,Y 113.963,Z 67.000,A 180.000,B 0.000,C 180.000} C_DIS
LIN {X 57.746,Y 113.977,Z 67.000,A 180.000,B 0.000,C 180.000} C_DIS
LIN {X 57.925,Y 113.983,Z 67.000,A 180.000,B 0.000,C 180.000} C_DIS
LIN {X 58.282,Y 113.994,Z 67.000,A 180.000,B 0.000,C 180.000} C_DIS
LIN {X 58.461,Y 114.000,Z 67.000,A 180.000,B 0.000,C 180.000} C_DIS
LIN {X 58.640,Y 113.997,Z 67.000,A 180.000,B 0.000,C 180.000} C_DIS
LIN {X 59.176,Y 113.980,Z 67.000,A 180.000,B 0.000,C 180.000} C_DIS
LIN {X 59.355,Y 113.970,Z 67.000,A 180.000,B 0.000,C 180.000} C_DIS
LIN {X 59.534,Y 113.953,Z 67.000,A 180.000,B 0.000,C 180.000} C_DIS
LIN {X 59.891,Y 113.919,Z 67.000,A 180.000,B 0.000,C 180.000} C_DIS
LIN {X 60.070,Y 113.901,Z 67.000,A 180.000,B 0.000,C 180.000} C_DIS
LIN {X 60.212,Y 113.880,Z 67.000,A 180.000,B 0.000,C 180.000} C_DIS
LIN {X 60.606,Y 113.817,Z 67.000,A 180.000,B 0.000,C 180.000} C_DIS
LIN {X 60.785,Y 113.789,Z 67.000,A 180.000,B 0.000,C 180.000} C_DIS
LIN {X 60.964,Y 113.753,Z 67.000,A 180.000,B 0.000,C 180.000} C_DIS
LIN {X 61.500,Y 113.633,Z 67.000,A 180.000,B 0.000,C 180.000} C_DIS
LIN {X 61.679,Y 113.588,Z 67.000,A 180.000,B 0.000,C 180.000} C_DIS
LIN {X 62.215,Y 113.432,Z 67.000,A 180.000,B 0.000,C 180.000} C_DIS
LIN {X 62.394,Y 113.378,Z 67.000,A 180.000,B 0.000,C 180.000} C_DIS
LIN {X 62.491,Y 113.343,Z 67.000,A 180.000,B 0.000,C 180.000} C_DIS
LIN {X 62.987,Y 113.165,Z 67.000,A 180.000,B 0.000,C 180.000} C_DIS
LIN {X 63.109,Y 113.119,Z 67.000,A 180.000,B 0.000,C 180.000} C_DIS
LIN {X 63.288,Y 113.043,Z 67.000,A 180.000,B 0.000,C 180.000} C_DIS
LIN {X 63.645,Y 112.888,Z 67.000,A 180.000,B 0.000,C 180.000} C_DIS
LIN {X 63.824,Y 112.809,Z 67.000,A 180.000,B 0.000,C 180.000} C_DIS
LIN {X 63.829,Y 112.807,Z 67.000,A 180.000,B 0.000,C 180.000} C_DIS
LIN {X 64.003,Y 112.720,Z 67.000,A 180.000,B 0.000,C 180.000} C_DIS
LIN {X 64.360,Y 112.538,Z 67.000,A 180.000,B 0.000,C 180.000} C_DIS
LIN {X 64.530,Y 112.450,Z 67.000,A 180.000,B 0.000,C 180.000} C_DIS
LIN {X 64.539,Y 112.444,Z 67.000,A 180.000,B 0.000,C 180.000} C_DIS
LIN {X 64.718,Y 112.339,Z 67.000,A 180.000,B 0.000,C 180.000} C_DIS
LIN {X 65.075,Y 112.128,Z 67.000,A 180.000,B 0.000,C 180.000} C_DIS
LIN {X 65.136,Y 112.092,Z 67.000,A 180.000,B 0.000,C 180.000} C_DIS
LIN {X 65.254,Y 112.017,Z 67.000,A 180.000,B 0.000,C 180.000} C_DIS
LIN {X 65.433,Y 111.896,Z 67.000,A 180.000,B 0.000,C 180.000} C_DIS
LIN {X 65.670,Y 111.734,Z 67.000,A 180.000,B 0.000,C 180.000} C_DIS
LIN {X 65.791,Y 111.653,Z 67.000,A 180.000,B 0.000,C 180.000} C_DIS
LIN {X 65.923,Y 111.556,Z 67.000,A 180.000,B 0.000,C 180.000} C_DIS
LIN {X 66.384,Y 111.198,Z 67.000,A 180.000,B 0.000,C 180.000} C_DIS
LIN {X 66.506,Y 111.099,Z 67.000,A 180.000,B 0.000,C 180.000} C_DIS
LIN {X 66.597,Y 111.019,Z 67.000,A 180.000,B 0.000,C 180.000} C_DIS
LIN {X 67.002,Y 110.662,Z 67.000,A 180.000,B 0.000,C 180.000} C_DIS
LIN {X 67.042,Y 110.626,Z 67.000,A 180.000,B 0.000,C 180.000} C_DIS
LIN {X 67.188,Y 110.483,Z 67.000,A 180.000,B 0.000,C 180.000} C_DIS
LIN {X 67.545,Y 110.126,Z 67.000,A 180.000,B 0.000,C 180.000} C_DIS
LIN {X 67.578,Y 110.092,Z 67.000,A 180.000,B 0.000,C 180.000} C_DIS
LIN {X 67.711,Y 109.947,Z 67.000,A 180.000,B 0.000,C 180.000} C_DIS
LIN {X 68.026,Y 109.589,Z 67.000,A 180.000,B 0.000,C 180.000} C_DIS
LIN {X 68.115,Y 109.488,Z 67.000,A 180.000,B 0.000,C 180.000} C_DIS
LIN {X 68.177,Y 109.410,Z 67.000,A 180.000,B 0.000,C 180.000} C_DIS
LIN {X 68.472,Y 109.031,Z 67.000,A 180.000,B 0.000,C 180.000} C_DIS
LIN {X 68.593,Y 108.874,Z 67.000,A 180.000,B 0.000,C 180.000} C_DIS
LIN {X 68.651,Y 108.793,Z 67.000,A 180.000,B 0.000,C 180.000} C_DIS
LIN {X 68.717,Y 108.695,Z 67.000,A 180.000,B 0.000,C 180.000} C_DIS
LIN {X 69.008,Y 108.267,Z 67.000,A 180.000,B 0.000,C 180.000} C_DIS
LIN {X 69.078,Y 108.159,Z 67.000,A 180.000,B 0.000,C 180.000} C_DIS
LIN {X 69.184,Y 107.980,Z 67.000,A 180.000,B 0.000,C 180.000} C_DIS
LIN {X 69.396,Y 107.623,Z 67.000,A 180.000,B 0.000,C 180.000} C_DIS
LIN {X 69.495,Y 107.444,Z 67.000,A 180.000,B 0.000,C 180.000} C_DIS
LIN {X 69.768,Y 106.908,Z 67.000,A 180.000,B 0.000,C 180.000} C_DIS
LIN {X 69.852,Y 106.729,Z 67.000,A 180.000,B 0.000,C 180.000} C_DIS
LIN {X 70.084,Y 106.193,Z 67.000,A 180.000,B 0.000,C 180.000} C_DIS
LIN {X 70.155,Y 106.014,Z 67.000,A 180.000,B 0.000,C 180.000} C_DIS
LIN {X 70.348,Y 105.477,Z 67.000,A 180.000,B 0.000,C 180.000} C_DIS
LIN {X 70.408,Y 105.299,Z 67.000,A 180.000,B 0.000,C 180.000} C_DIS
LIN {X 70.439,Y 105.194,Z 67.000,A 180.000,B 0.000,C 180.000} C_DIS
LIN {X 70.564,Y 104.762,Z 67.000,A 180.000,B 0.000,C 180.000} C_DIS
LIN {X 70.614,Y 104.584,Z 67.000,A 180.000,B 0.000,C 180.000} C_DIS
LIN {X 70.617,Y 104.568,Z 67.000,A 180.000,B 0.000,C 180.000} C_DIS
LIN {X 70.654,Y 104.405,Z 67.000,A 180.000,B 0.000,C 180.000} C_DIS
LIN {X 70.734,Y 104.047,Z 67.000,A 180.000,B 0.000,C 180.000} C_DIS
LIN {X 70.773,Y 103.869,Z 67.000,A 180.000,B 0.000,C 180.000} C_DIS
LIN {X 70.796,Y 103.739,Z 67.000,A 180.000,B 0.000,C 180.000} C_DIS
LIN {X 70.889,Y 103.153,Z 67.000,A 180.000,B 0.000,C 180.000} C_DIS
LIN {X 70.911,Y 102.975,Z 67.000,A 180.000,B 0.000,C 180.000} C_DIS
LIN {X 70.962,Y 102.438,Z 67.000,A 180.000,B 0.000,C 180.000} C_DIS
LIN {X 70.975,Y 102.292,Z 67.000,A 180.000,B 0.000,C 180.000} C_DIS
LIN {X 70.977,Y 102.260,Z 67.000,A 180.000,B 0.000,C 180.000} C_DIS
LIN {X 70.983,Y 102.081,Z 67.000,A 180.000,B 0.000,C 180.000} C_DIS
LIN {X 70.994,Y 101.723,Z 67.000,A 180.000,B 0.000,C 180.000} C_DIS
LIN {X 71.000,Y 101.545,Z 67.000,A 180.000,B 0.000,C 180.000} C_DIS
LIN {X 70.997,Y 101.366,Z 67.000,A 180.000,B 0.000,C 180.000} C_DIS
LIN {X 70.980,Y 100.829,Z 67.000,A 180.000,B 0.000,C 180.000} C_DIS
LIN {X 70.975,Y 100.708,Z 67.000,A 180.000,B 0.000,C 180.000} C_DIS
LIN {X 70.970,Y 100.651,Z 67.000,A 180.000,B 0.000,C 180.000} C_DIS
LIN {X 70.954,Y 100.472,Z 67.000,A 180.000,B 0.000,C 180.000} C_DIS
LIN {X 70.920,Y 100.114,Z 67.000,A 180.000,B 0.000,C 180.000} C_DIS
LIN {X 70.902,Y 99.936,Z 67.000,A 180.000,B 0.000,C 180.000} C_DIS
LIN {X 70.875,Y 99.757,Z 67.000,A 180.000,B 0.000,C 180.000} C_DIS
LIN {X 70.796,Y 99.261,Z 67.000,A 180.000,B 0.000,C 180.000} C_DIS
LIN {X 70.790,Y 99.221,Z 67.000,A 180.000,B 0.000,C 180.000} C_DIS
LIN {X 70.754,Y 99.042,Z 67.000,A 180.000,B 0.000,C 180.000} C_DIS
LIN {X 70.670,Y 98.665,Z 67.000,A 180.000,B 0.000,C 180.000} C_DIS
LIN {X 70.634,Y 98.505,Z 67.000,A 180.000,B 0.000,C 180.000} C_DIS
LIN {X 70.617,Y 98.432,Z 67.000,A 180.000,B 0.000,C 180.000} C_DIS
LIN {X 70.590,Y 98.327,Z 67.000,A 180.000,B 0.000,C 180.000} C_DIS
LIN {X 70.538,Y 98.148,Z 67.000,A 180.000,B 0.000,C 180.000} C_DIS
LIN {X 70.434,Y 97.790,Z 67.000,A 180.000,B 0.000,C 180.000} C_DIS
LIN {X 70.380,Y 97.612,Z 67.000,A 180.000,B 0.000,C 180.000} C_DIS
LIN {X 70.316,Y 97.433,Z 67.000,A 180.000,B 0.000,C 180.000} C_DIS
LIN {X 70.187,Y 97.075,Z 67.000,A 180.000,B 0.000,C 180.000} C_DIS
LIN {X 70.121,Y 96.897,Z 67.000,A 180.000,B 0.000,C 180.000} C_DIS
LIN {X 70.081,Y 96.800,Z 67.000,A 180.000,B 0.000,C 180.000} C_DIS
LIN {X 69.891,Y 96.360,Z 67.000,A 180.000,B 0.000,C 180.000} C_DIS
LIN {X 69.812,Y 96.181,Z 67.000,A 180.000,B 0.000,C 180.000} C_DIS
LIN {X 69.724,Y 96.005,Z 67.000,A 180.000,B 0.000,C 180.000} C_DIS
LIN {X 69.540,Y 95.645,Z 67.000,A 180.000,B 0.000,C 180.000} C_DIS
LIN {X 69.447,Y 95.466,Z 67.000,A 180.000,B 0.000,C 180.000} C_DIS
LIN {X 69.366,Y 95.327,Z 67.000,A 180.000,B 0.000,C 180.000} C_DIS
LIN {X 69.131,Y 94.930,Z 67.000,A 180.000,B 0.000,C 180.000} C_DIS
LIN {X 69.021,Y 94.751,Z 67.000,A 180.000,B 0.000,C 180.000} C_DIS
LIN {X 69.008,Y 94.733,Z 67.000,A 180.000,B 0.000,C 180.000} C_DIS
LIN {X 68.657,Y 94.215,Z 67.000,A 180.000,B 0.000,C 180.000} C_DIS
LIN {X 68.651,Y 94.207,Z 67.000,A 180.000,B 0.000,C 180.000} C_DIS
LIN {X 68.524,Y 94.036,Z 67.000,A 180.000,B 0.000,C 180.000} C_DIS
LIN {X 68.247,Y 93.679,Z 67.000,A 180.000,B 0.000,C 180.000} C_DIS
LIN {X 68.115,Y 93.512,Z 67.000,A 180.000,B 0.000,C 180.000} C_DIS
LIN {X 68.104,Y 93.500,Z 67.000,A 180.000,B 0.000,C 180.000} C_DIS
LIN {X 67.947,Y 93.321,Z 67.000,A 180.000,B 0.000,C 180.000} C_DIS
LIN {X 67.757,Y 93.106,Z 67.000,A 180.000,B 0.000,C 180.000} C_DIS
LIN {X 67.631,Y 92.964,Z 67.000,A 180.000,B 0.000,C 180.000} C_DIS
LIN {X 67.578,Y 92.908,Z 67.000,A 180.000,B 0.000,C 180.000} C_DIS
LIN {X 67.456,Y 92.785,Z 67.000,A 180.000,B 0.000,C 180.000} C_DIS
LIN {X 67.221,Y 92.550,Z 67.000,A 180.000,B 0.000,C 180.000} C_DIS
LIN {X 67.098,Y 92.427,Z 67.000,A 180.000,B 0.000,C 180.000} C_DIS
LIN {X 67.042,Y 92.374,Z 67.000,A 180.000,B 0.000,C 180.000} C_DIS
LIN {X 66.901,Y 92.249,Z 67.000,A 180.000,B 0.000,C 180.000} C_DIS
LIN {X 66.684,Y 92.058,Z 67.000,A 180.000,B 0.000,C 180.000} C_DIS
LIN {X 66.506,Y 91.901,Z 67.000,A 180.000,B 0.000,C 180.000} C_DIS
LIN {X 66.494,Y 91.891,Z 67.000,A 180.000,B 0.000,C 180.000} C_DIS
LIN {X 66.327,Y 91.758,Z 67.000,A 180.000,B 0.000,C 180.000} C_DIS
LIN {X 65.969,Y 91.480,Z 67.000,A 180.000,B 0.000,C 180.000} C_DIS
LIN {X 65.801,Y 91.355,Z 67.000,A 180.000,B 0.000,C 180.000} C_DIS
LIN {X 65.791,Y 91.347,Z 67.000,A 180.000,B 0.000,C 180.000} C_DIS
LIN {X 65.538,Y 91.176,Z 67.000,A 180.000,B 0.000,C 180.000} C_DIS
LIN {X 65.275,Y 90.997,Z 67.000,A 180.000,B 0.000,C 180.000} C_DIS
LIN {X 65.254,Y 90.983,Z 67.000,A 180.000,B 0.000,C 180.000} C_DIS
LIN {X 65.075,Y 90.872,Z 67.000,A 180.000,B 0.000,C 180.000} C_DIS
LIN {X 64.682,Y 90.640,Z 67.000,A 180.000,B 0.000,C 180.000} C_DIS
LIN {X 64.539,Y 90.556,Z 67.000,A 180.000,B 0.000,C 180.000} C_DIS
LIN {X 64.360,Y 90.462,Z 67.000,A 180.000,B 0.000,C 180.000} C_DIS
LIN {X 64.003,Y 90.280,Z 67.000,A 180.000,B 0.000,C 180.000} C_DIS
LIN {X 63.824,Y 90.191,Z 67.000,A 180.000,B 0.000,C 180.000} C_DIS
LIN {X 63.645,Y 90.112,Z 67.000,A 180.000,B 0.000,C 180.000} C_DIS
LIN {X 63.213,Y 89.925,Z 67.000,A 180.000,B 0.000,C 180.000} C_DIS
LIN {X 63.109,Y 89.881,Z 67.000,A 180.000,B 0.000,C 180.000} C_DIS
LIN {X 62.930,Y 89.815,Z 67.000,A 180.000,B 0.000,C 180.000} C_DIS
LIN {X 62.573,Y 89.686,Z 67.000,A 180.000,B 0.000,C 180.000} C_DIS
LIN {X 62.394,Y 89.622,Z 67.000,A 180.000,B 0.000,C 180.000} C_DIS
LIN {X 62.215,Y 89.568,Z 67.000,A 180.000,B 0.000,C 180.000} C_DIS
LIN {X 61.679,Y 89.412,Z 67.000,A 180.000,B 0.000,C 180.000} C_DIS
LIN {X 61.591,Y 89.388,Z 67.000,A 180.000,B 0.000,C 180.000} C_DIS
LIN {X 61.500,Y 89.367,Z 67.000,A 180.000,B 0.000,C 180.000} C_DIS
LIN {X 60.964,Y 89.247,Z 67.000,A 180.000,B 0.000,C 180.000} C_DIS
LIN {X 60.785,Y 89.211,Z 67.000,A 180.000,B 0.000,C 180.000} C_DIS
LIN {X 60.774,Y 89.209,Z 67.000,A 180.000,B 0.000,C 180.000} C_DIS
LIN {X 60.606,Y 89.183,Z 67.000,A 180.000,B 0.000,C 180.000} C_DIS
LIN {X 60.249,Y 89.126,Z 67.000,A 180.000,B 0.000,C 180.000} C_DIS
LIN {X 60.070,Y 89.099,Z 67.000,A 180.000,B 0.000,C 180.000} C_DIS
LIN {X 59.891,Y 89.081,Z 67.000,A 180.000,B 0.000,C 180.000} C_DIS
LIN {X 59.361,Y 89.031,Z 67.000,A 180.000,B 0.000,C 180.000} C_DIS
LIN {X 59.355,Y 89.030,Z 67.000,A 180.000,B 0.000,C 180.000} C_DIS
LIN {X 59.176,Y 89.020,Z 67.000,A 180.000,B 0.000,C 180.000} C_DIS
LIN {X 58.640,Y 89.003,Z 67.000,A 180.000,B 0.000,C 180.000} C_DIS
LIN {X 58.461,Y 89.000,Z 67.000,A 180.000,B 0.000,C 180.000} C_DIS
LIN {X 58.282,Y 89.006,Z 67.000,A 180.000,B 0.000,C 180.000} C_DIS
LIN {X 57.925,Y 89.017,Z 67.000,A 180.000,B 0.000,C 180.000} C_DIS
LIN {X 57.746,Y 89.023,Z 67.000,A 180.000,B 0.000,C 180.000} C_DIS
LIN {X 57.639,Y 89.031,Z 67.000,A 180.000,B 0.000,C 180.000} C_DIS
LIN {X 57.031,Y 89.088,Z 67.000,A 180.000,B 0.000,C 180.000} C_DIS
LIN {X 56.852,Y 89.110,Z 67.000,A 180.000,B 0.000,C 180.000} C_DIS
LIN {X 56.316,Y 89.195,Z 67.000,A 180.000,B 0.000,C 180.000} C_DIS
LIN {X 56.226,Y 89.209,Z 67.000,A 180.000,B 0.000,C 180.000} C_DIS
LIN {X 56.137,Y 89.225,Z 67.000,A 180.000,B 0.000,C 180.000} C_DIS
LIN {X 55.958,Y 89.265,Z 67.000,A 180.000,B 0.000,C 180.000} C_DIS
LIN {X 55.601,Y 89.345,Z 67.000,A 180.000,B 0.000,C 180.000} C_DIS
LIN {X 55.422,Y 89.385,Z 67.000,A 180.000,B 0.000,C 180.000} C_DIS
LIN {X 55.409,Y 89.388,Z 67.000,A 180.000,B 0.000,C 180.000} C_DIS
LIN {X 55.243,Y 89.434,Z 67.000,A 180.000,B 0.000,C 180.000} C_DIS
LIN {X 54.787,Y 89.567,Z 67.000,A 180.000,B 0.000,C 180.000} C_DIS
LIN {X 54.707,Y 89.590,Z 67.000,A 180.000,B 0.000,C 180.000} C_DIS
LIN {X 54.528,Y 89.650,Z 67.000,A 180.000,B 0.000,C 180.000} C_DIS
LIN {X 53.992,Y 89.843,Z 67.000,A 180.000,B 0.000,C 180.000} C_DIS
LIN {X 53.813,Y 89.913,Z 67.000,A 180.000,B 0.000,C 180.000} C_DIS
LIN {X 53.277,Y 90.146,Z 67.000,A 180.000,B 0.000,C 180.000} C_DIS
LIN {X 53.098,Y 90.229,Z 67.000,A 180.000,B 0.000,C 180.000} C_DIS
LIN {X 52.562,Y 90.502,Z 67.000,A 180.000,B 0.000,C 180.000} C_DIS
LIN {X 52.383,Y 90.601,Z 67.000,A 180.000,B 0.000,C 180.000} C_DIS
LIN {X 52.015,Y 90.818,Z 67.000,A 180.000,B 0.000,C 180.000} C_DIS
LIN {X 51.847,Y 90.918,Z 67.000,A 180.000,B 0.000,C 180.000} C_DIS
LIN {X 51.725,Y 90.997,Z 67.000,A 180.000,B 0.000,C 180.000} C_DIS
LIN {X 51.310,Y 91.279,Z 67.000,A 180.000,B 0.000,C 180.000} C_DIS
LIN {X 51.199,Y 91.355,Z 67.000,A 180.000,B 0.000,C 180.000} C_DIS
LIN {X 51.131,Y 91.403,Z 67.000,A 180.000,B 0.000,C 180.000} C_DIS
LIN {X 50.962,Y 91.533,Z 67.000,A 180.000,B 0.000,C 180.000} C_DIS
LIN {X 50.595,Y 91.818,Z 67.000,A 180.000,B 0.000,C 180.000} C_DIS
LIN {X 50.506,Y 91.891,Z 67.000,A 180.000,B 0.000,C 180.000} C_DIS
LIN {X 50.416,Y 91.969,Z 67.000,A 180.000,B 0.000,C 180.000} C_DIS
LIN {X 50.059,Y 92.284,Z 67.000,A 180.000,B 0.000,C 180.000} C_DIS
LIN {X 49.902,Y 92.427,Z 67.000,A 180.000,B 0.000,C 180.000} C_DIS
LIN {X 49.880,Y 92.449,Z 67.000,A 180.000,B 0.000,C 180.000} C_DIS
LIN {X 49.523,Y 92.807,Z 67.000,A 180.000,B 0.000,C 180.000} C_DIS
LIN {X 49.369,Y 92.964,Z 67.000,A 180.000,B 0.000,C 180.000} C_DIS
LIN {X 49.344,Y 92.991,Z 67.000,A 180.000,B 0.000,C 180.000} C_DIS
LIN {X 49.211,Y 93.142,Z 67.000,A 180.000,B 0.000,C 180.000} C_DIS
LIN {X 48.986,Y 93.397,Z 67.000,A 180.000,B 0.000,C 180.000} C_DIS
LIN {X 48.896,Y 93.500,Z 67.000,A 180.000,B 0.000,C 180.000} C_DIS
LIN {X 48.807,Y 93.609,Z 67.000,A 180.000,B 0.000,C 180.000} C_DIS
LIN {X 48.450,Y 94.070,Z 67.000,A 180.000,B 0.000,C 180.000} C_DIS
LIN {X 48.343,Y 94.215,Z 67.000,A 180.000,B 0.000,C 180.000} C_DIS
LIN {X 48.092,Y 94.584,Z 67.000,A 180.000,B 0.000,C 180.000} C_DIS
LIN {X 47.979,Y 94.751,Z 67.000,A 180.000,B 0.000,C 180.000} C_DIS
LIN {X 47.914,Y 94.855,Z 67.000,A 180.000,B 0.000,C 180.000} C_DIS
LIN {X 47.869,Y 94.930,Z 67.000,A 180.000,B 0.000,C 180.000} C_DIS
LIN {X 47.657,Y 95.288,Z 67.000,A 180.000,B 0.000,C 180.000} C_DIS
LIN {X 47.556,Y 95.460,Z 67.000,A 180.000,B 0.000,C 180.000} C_DIS
LIN {X 47.553,Y 95.466,Z 67.000,A 180.000,B 0.000,C 180.000} C_DIS
LIN {X 47.460,Y 95.645,Z 67.000,A 180.000,B 0.000,C 180.000} C_DIS
LIN {X 47.277,Y 96.003,Z 67.000,A 180.000,B 0.000,C 180.000} C_DIS
LIN {X 47.198,Y 96.159,Z 67.000,A 180.000,B 0.000,C 180.000} C_DIS
LIN {X 47.188,Y 96.181,Z 67.000,A 180.000,B 0.000,C 180.000} C_DIS
LIN {X 47.109,Y 96.360,Z 67.000,A 180.000,B 0.000,C 180.000} C_DIS
LIN {X 46.955,Y 96.718,Z 67.000,A 180.000,B 0.000,C 180.000} C_DIS
LIN {X 46.879,Y 96.897,Z 67.000,A 180.000,B 0.000,C 180.000} C_DIS
LIN {X 46.841,Y 96.997,Z 67.000,A 180.000,B 0.000,C 180.000} C_DIS
LIN {X 46.662,Y 97.494,Z 67.000,A 180.000,B 0.000,C 180.000} C_DIS
LIN {X 46.620,Y 97.612,Z 67.000,A 180.000,B 0.000,C 180.000} C_DIS
LIN {X 46.566,Y 97.790,Z 67.000,A 180.000,B 0.000,C 180.000} C_DIS
LIN {X 46.462,Y 98.148,Z 67.000,A 180.000,B 0.000,C 180.000} C_DIS
LIN {X 46.410,Y 98.327,Z 67.000,A 180.000,B 0.000,C 180.000} C_DIS
LIN {X 46.366,Y 98.505,Z 67.000,A 180.000,B 0.000,C 180.000} C_DIS
LIN {X 46.246,Y 99.042,Z 67.000,A 180.000,B 0.000,C 180.000} C_DIS
LIN {X 46.210,Y 99.221,Z 67.000,A 180.000,B 0.000,C 180.000} C_DIS
LIN {X 46.182,Y 99.399,Z 67.000,A 180.000,B 0.000,C 180.000} C_DIS
LIN {X 46.126,Y 99.753,Z 67.000,A 180.000,B 0.000,C 180.000} C_DIS
LIN {X 46.125,Y 99.757,Z 67.000,A 180.000,B 0.000,C 180.000} C_DIS
LIN {X 46.098,Y 99.936,Z 67.000,A 180.000,B 0.000,C 180.000} C_DIS
LIN {X 46.080,Y 100.114,Z 67.000,A 180.000,B 0.000,C 180.000} C_DIS
LIN {X 46.077,Y 100.144,Z 67.000,A 180.000,B 0.000,C 180.000} C_DIS
; Link Move Starts
LIN {X 46.048,Y 100.458,Z 67.000,A 180.000,B 0.000,C 180.000} C_DIS
LIN {X 46.022,Y 100.772,Z 66.998,A 180.000,B 0.000,C 180.000} C_DIS
LIN {X 46.012,Y 101.087,Z 66.996,A 180.000,B 0.000,C 180.000} C_DIS
LIN {X 46.002,Y 101.401,Z 66.992,A 180.000,B 0.000,C 180.000} C_DIS
LIN {X 46.006,Y 101.716,Z 66.988,A 180.000,B 0.000,C 180.000} C_DIS
LIN {X 46.015,Y 102.031,Z 66.983,A 180.000,B 0.000,C 180.000} C_DIS
LIN {X 46.020,Y 102.189,Z 66.981,A 180.000,B 0.000,C 180.000} C_DIS
LIN {X 46.029,Y 102.346,Z 66.978,A 180.000,B 0.000,C 180.000} C_DIS
LIN {X 46.044,Y 102.503,Z 66.975,A 180.000,B 0.000,C 180.000} C_DIS
LIN {X 46.059,Y 102.659,Z 66.971,A 180.000,B 0.000,C 180.000} C_DIS
LIN {X 46.074,Y 102.816,Z 66.968,A 180.000,B 0.000,C 180.000} C_DIS
LIN {X 46.088,Y 102.973,Z 66.964,A 180.000,B 0.000,C 180.000} C_DIS
LIN {X 46.107,Y 103.129,Z 66.960,A 180.000,B 0.000,C 180.000} C_DIS
LIN {X 46.132,Y 103.285,Z 66.956,A 180.000,B 0.000,C 180.000} C_DIS
LIN {X 46.157,Y 103.441,Z 66.952,A 180.000,B 0.000,C 180.000} C_DIS
LIN {X 46.181,Y 103.596,Z 66.948,A 180.000,B 0.000,C 180.000} C_DIS
LIN {X 46.206,Y 103.752,Z 66.944,A 180.000,B 0.000,C 180.000} C_DIS
LIN {X 46.235,Y 103.907,Z 66.939,A 180.000,B 0.000,C 180.000} C_DIS
LIN {X 46.269,Y 104.060,Z 66.934,A 180.000,B 0.000,C 180.000} C_DIS
LIN {X 46.303,Y 104.214,Z 66.929,A 180.000,B 0.000,C 180.000} C_DIS
LIN {X 46.338,Y 104.368,Z 66.924,A 180.000,B 0.000,C 180.000} C_DIS
LIN {X 46.355,Y 104.445,Z 66.922,A 180.000,B 0.000,C 180.000} C_DIS
LIN {X 46.372,Y 104.521,Z 66.919,A 180.000,B 0.000,C 180.000} C_DIS
LIN {X 46.390,Y 104.598,Z 66.917,A 180.000,B 0.000,C 180.000} C_DIS
LIN {X 46.410,Y 104.674,Z 66.914,A 180.000,B 0.000,C 180.000} C_DIS
LIN {X 46.432,Y 104.750,Z 66.911,A 180.000,B 0.000,C 180.000} C_DIS
LIN {X 46.454,Y 104.825,Z 66.909,A 180.000,B 0.000,C 180.000} C_DIS
LIN {X 46.476,Y 104.901,Z 66.906,A 180.000,B 0.000,C 180.000} C_DIS
LIN {X 46.498,Y 104.977,Z 66.903,A 180.000,B 0.000,C 180.000} C_DIS
LIN {X 46.520,Y 105.052,Z 66.901,A 180.000,B 0.000,C 180.000} C_DIS
LIN {X 46.542,Y 105.128,Z 66.898,A 180.000,B 0.000,C 180.000} C_DIS
LIN {X 46.564,Y 105.203,Z 66.895,A 180.000,B 0.000,C 180.000} C_DIS
LIN {X 46.586,Y 105.279,Z 66.892,A 180.000,B 0.000,C 180.000} C_DIS
LIN {X 46.609,Y 105.354,Z 66.890,A 180.000,B 0.000,C 180.000} C_DIS
LIN {X 46.634,Y 105.429,Z 66.887,A 180.000,B 0.000,C 180.000} C_DIS
LIN {X 46.661,Y 105.503,Z 66.884,A 180.000,B 0.000,C 180.000} C_DIS
LIN {X 46.688,Y 105.577,Z 66.881,A 180.000,B 0.000,C 180.000} C_DIS
LIN {X 46.714,Y 105.651,Z 66.878,A 180.000,B 0.000,C 180.000} C_DIS
LIN {X 46.741,Y 105.725,Z 66.876,A 180.000,B 0.000,C 180.000} C_DIS
LIN {X 46.768,Y 105.800,Z 66.873,A 180.000,B 0.000,C 180.000} C_DIS
LIN {X 46.794,Y 105.874,Z 66.870,A 180.000,B 0.000,C 180.000} C_DIS
LIN {X 46.821,Y 105.948,Z 66.867,A 180.000,B 0.000,C 180.000} C_DIS
LIN {X 46.848,Y 106.022,Z 66.865,A 180.000,B 0.000,C 180.000} C_DIS
LIN {X 46.875,Y 106.096,Z 66.862,A 180.000,B 0.000,C 180.000} C_DIS
LIN {X 46.905,Y 106.168,Z 66.859,A 180.000,B 0.000,C 180.000} C_DIS
LIN {X 46.937,Y 106.241,Z 66.856,A 180.000,B 0.000,C 180.000} C_DIS
LIN {X 46.968,Y 106.313,Z 66.854,A 180.000,B 0.000,C 180.000} C_DIS
LIN {X 47.030,Y 106.458,Z 66.848,A 180.000,B 0.000,C 180.000} C_DIS
LIN {X 47.124,Y 106.674,Z 66.840,A 180.000,B 0.000,C 180.000} C_DIS
LIN {X 47.156,Y 106.747,Z 66.837,A 180.000,B 0.000,C 180.000} C_DIS
LIN {X 47.188,Y 106.818,Z 66.834,A 180.000,B 0.000,C 180.000} C_DIS
LIN {X 47.222,Y 106.889,Z 66.832,A 180.000,B 0.000,C 180.000} C_DIS
LIN {X 47.294,Y 107.030,Z 66.826,A 180.000,B 0.000,C 180.000} C_DIS
LIN {X 47.401,Y 107.240,Z 66.818,A 180.000,B 0.000,C 180.000} C_DIS
LIN {X 47.473,Y 107.380,Z 66.812,A 180.000,B 0.000,C 180.000} C_DIS
LIN {X 47.508,Y 107.451,Z 66.810,A 180.000,B 0.000,C 180.000} C_DIS
LIN {X 47.545,Y 107.520,Z 66.807,A 180.000,B 0.000,C 180.000} C_DIS
LIN {X 47.584,Y 107.589,Z 66.804,A 180.000,B 0.000,C 180.000} C_DIS
LIN {X 47.825,Y 107.995,Z 66.788,A 180.000,B 0.000,C 180.000} C_DIS
LIN {X 47.905,Y 108.131,Z 66.782,A 180.000,B 0.000,C 180.000} C_DIS
LIN {X 47.946,Y 108.198,Z 66.779,A 180.000,B 0.000,C 180.000} C_DIS
LIN {X 47.989,Y 108.264,Z 66.777,A 180.000,B 0.000,C 180.000} C_DIS
LIN {X 48.166,Y 108.524,Z 66.766,A 180.000,B 0.000,C 180.000} C_DIS
LIN {X 48.343,Y 108.785,Z 66.755,A 180.000,B 0.000,C 180.000} C_DIS
LIN {X 48.389,Y 108.849,Z 66.752,A 180.000,B 0.000,C 180.000} C_DIS
LIN {X 48.436,Y 108.912,Z 66.749,A 180.000,B 0.000,C 180.000} C_DIS
LIN {X 48.822,Y 109.410,Z 66.727,A 180.000,B 0.000,C 180.000} C_DIS
LIN {X 48.872,Y 109.471,Z 66.724,A 180.000,B 0.000,C 180.000} C_DIS
LIN {X 48.923,Y 109.531,Z 66.722,A 180.000,B 0.000,C 180.000} C_DIS
LIN {X 49.079,Y 109.708,Z 66.713,A 180.000,B 0.000,C 180.000} C_DIS
LIN {X 49.183,Y 109.827,Z 66.708,A 180.000,B 0.000,C 180.000} C_DIS
LIN {X 49.287,Y 109.945,Z 66.702,A 180.000,B 0.000,C 180.000} C_DIS
LIN {X 49.339,Y 110.004,Z 66.700,A 180.000,B 0.000,C 180.000} C_DIS
LIN {X 49.393,Y 110.062,Z 66.697,A 180.000,B 0.000,C 180.000} C_DIS
LIN {X 49.448,Y 110.118,Z 66.694,A 180.000,B 0.000,C 180.000} C_DIS
LIN {X 49.615,Y 110.285,Z 66.686,A 180.000,B 0.000,C 180.000} C_DIS
LIN {X 49.726,Y 110.397,Z 66.680,A 180.000,B 0.000,C 180.000} C_DIS
LIN {X 49.782,Y 110.452,Z 66.678,A 180.000,B 0.000,C 180.000} C_DIS
LIN {X 49.837,Y 110.508,Z 66.675,A 180.000,B 0.000,C 180.000} C_DIS
LIN {X 49.893,Y 110.564,Z 66.672,A 180.000,B 0.000,C 180.000} C_DIS
LIN {X 49.950,Y 110.618,Z 66.669,A 180.000,B 0.000,C 180.000} C_DIS
LIN {X 50.008,Y 110.671,Z 66.667,A 180.000,B 0.000,C 180.000} C_DIS
LIN {X 50.126,Y 110.775,Z 66.661,A 180.000,B 0.000,C 180.000} C_DIS
LIN {X 50.304,Y 110.932,Z 66.653,A 180.000,B 0.000,C 180.000} C_DIS
LIN {X 50.422,Y 111.036,Z 66.647,A 180.000,B 0.000,C 180.000} C_DIS
LIN {X 50.481,Y 111.088,Z 66.645,A 180.000,B 0.000,C 180.000} C_DIS
LIN {X 50.541,Y 111.139,Z 66.642,A 180.000,B 0.000,C 180.000} C_DIS
LIN {X 50.603,Y 111.188,Z 66.639,A 180.000,B 0.000,C 180.000} C_DIS
LIN {X 50.665,Y 111.236,Z 66.636,A 180.000,B 0.000,C 180.000} C_DIS
LIN {X 50.727,Y 111.284,Z 66.634,A 180.000,B 0.000,C 180.000} C_DIS
LIN {X 50.789,Y 111.332,Z 66.631,A 180.000,B 0.000,C 180.000} C_DIS
LIN {X 50.852,Y 111.381,Z 66.628,A 180.000,B 0.000,C 180.000} C_DIS
LIN {X 50.914,Y 111.429,Z 66.625,A 180.000,B 0.000,C 180.000} C_DIS
LIN {X 50.976,Y 111.477,Z 66.623,A 180.000,B 0.000,C 180.000} C_DIS
LIN {X 51.038,Y 111.526,Z 66.620,A 180.000,B 0.000,C 180.000} C_DIS
LIN {X 51.101,Y 111.574,Z 66.617,A 180.000,B 0.000,C 180.000} C_DIS
LIN {X 51.164,Y 111.621,Z 66.614,A 180.000,B 0.000,C 180.000} C_DIS
LIN {X 51.228,Y 111.666,Z 66.612,A 180.000,B 0.000,C 180.000} C_DIS
LIN {X 51.294,Y 111.710,Z 66.609,A 180.000,B 0.000,C 180.000} C_DIS
LIN {X 51.359,Y 111.754,Z 66.606,A 180.000,B 0.000,C 180.000} C_DIS
LIN {X 51.424,Y 111.798,Z 66.603,A 180.000,B 0.000,C 180.000} C_DIS
LIN {X 51.489,Y 111.843,Z 66.601,A 180.000,B 0.000,C 180.000} C_DIS
LIN {X 51.554,Y 111.887,Z 66.598,A 180.000,B 0.000,C 180.000} C_DIS
LIN {X 51.619,Y 111.931,Z 66.595,A 180.000,B 0.000,C 180.000} C_DIS
LIN {X 51.684,Y 111.976,Z 66.592,A 180.000,B 0.000,C 180.000} C_DIS
LIN {X 51.750,Y 112.020,Z 66.590,A 180.000,B 0.000,C 180.000} C_DIS
LIN {X 51.816,Y 112.063,Z 66.587,A 180.000,B 0.000,C 180.000} C_DIS
LIN {X 51.883,Y 112.103,Z 66.584,A 180.000,B 0.000,C 180.000} C_DIS
LIN {X 51.951,Y 112.143,Z 66.582,A 180.000,B 0.000,C 180.000} C_DIS
LIN {X 52.019,Y 112.184,Z 66.579,A 180.000,B 0.000,C 180.000} C_DIS
LIN {X 52.086,Y 112.224,Z 66.577,A 180.000,B 0.000,C 180.000} C_DIS
LIN {X 52.154,Y 112.264,Z 66.574,A 180.000,B 0.000,C 180.000} C_DIS
LIN {X 52.290,Y 112.344,Z 66.569,A 180.000,B 0.000,C 180.000} C_DIS
LIN {X 52.425,Y 112.424,Z 66.564,A 180.000,B 0.000,C 180.000} C_DIS
LIN {X 52.564,Y 112.499,Z 66.560,A 180.000,B 0.000,C 180.000} C_DIS
LIN {X 52.704,Y 112.570,Z 66.555,A 180.000,B 0.000,C 180.000} C_DIS
LIN {X 52.844,Y 112.642,Z 66.551,A 180.000,B 0.000,C 180.000} C_DIS
LIN {X 52.985,Y 112.713,Z 66.547,A 180.000,B 0.000,C 180.000} C_DIS
LIN {X 53.125,Y 112.785,Z 66.542,A 180.000,B 0.000,C 180.000} C_DIS
LIN {X 53.268,Y 112.851,Z 66.539,A 180.000,B 0.000,C 180.000} C_DIS
LIN {X 53.413,Y 112.913,Z 66.535,A 180.000,B 0.000,C 180.000} C_DIS
LIN {X 53.557,Y 112.976,Z 66.531,A 180.000,B 0.000,C 180.000} C_DIS
LIN {X 53.702,Y 113.038,Z 66.528,A 180.000,B 0.000,C 180.000} C_DIS
LIN {X 53.846,Y 113.101,Z 66.524,A 180.000,B 0.000,C 180.000} C_DIS
LIN {X 53.993,Y 113.158,Z 66.521,A 180.000,B 0.000,C 180.000} C_DIS
LIN {X 54.142,Y 113.211,Z 66.519,A 180.000,B 0.000,C 180.000} C_DIS
LIN {X 54.290,Y 113.264,Z 66.516,A 180.000,B 0.000,C 180.000} C_DIS
LIN {X 54.586,Y 113.371,Z 66.511,A 180.000,B 0.000,C 180.000} C_DIS
LIN {X 54.888,Y 113.462,Z 66.507,A 180.000,B 0.000,C 180.000} C_DIS
LIN {X 55.190,Y 113.550,Z 66.504,A 180.000,B 0.000,C 180.000} C_DIS
LIN {X 55.494,Y 113.632,Z 66.502,A 180.000,B 0.000,C 180.000} C_DIS
LIN {X 55.802,Y 113.700,Z 66.500,A 180.000,B 0.000,C 180.000} C_DIS
LIN {X 56.066,Y 113.759,Z 66.500,A 180.000,B 0.000,C 180.000} C_DIS
; Cutting Move Starts
LIN {X 56.137,Y 113.775,Z 66.500,A 180.000,B 0.000,C 180.000} C_DIS
LIN {X 56.316,Y 113.805,Z 66.500,A 180.000,B 0.000,C 180.000} C_DIS
LIN {X 56.852,Y 113.890,Z 66.500,A 180.000,B 0.000,C 180.000} C_DIS
LIN {X 57.031,Y 113.912,Z 66.500,A 180.000,B 0.000,C 180.000} C_DIS
LIN {X 57.567,Y 113.963,Z 66.500,A 180.000,B 0.000,C 180.000} C_DIS
LIN {X 57.746,Y 113.977,Z 66.500,A 180.000,B 0.000,C 180.000} C_DIS
LIN {X 57.925,Y 113.983,Z 66.500,A 180.000,B 0.000,C 180.000} C_DIS
LIN {X 58.282,Y 113.994,Z 66.500,A 180.000,B 0.000,C 180.000} C_DIS
LIN {X 58.461,Y 114.000,Z 66.500,A 180.000,B 0.000,C 180.000} C_DIS
LIN {X 58.640,Y 113.997,Z 66.500,A 180.000,B 0.000,C 180.000} C_DIS
LIN {X 59.176,Y 113.980,Z 66.500,A 180.000,B 0.000,C 180.000} C_DIS
LIN {X 59.355,Y 113.970,Z 66.500,A 180.000,B 0.000,C 180.000} C_DIS
LIN {X 59.534,Y 113.953,Z 66.500,A 180.000,B 0.000,C 180.000} C_DIS
LIN {X 59.891,Y 113.919,Z 66.500,A 180.000,B 0.000,C 180.000} C_DIS
LIN {X 60.070,Y 113.901,Z 66.500,A 180.000,B 0.000,C 180.000} C_DIS
LIN {X 60.212,Y 113.880,Z 66.500,A 180.000,B 0.000,C 180.000} C_DIS
LIN {X 60.606,Y 113.817,Z 66.500,A 180.000,B 0.000,C 180.000} C_DIS
LIN {X 60.785,Y 113.789,Z 66.500,A 180.000,B 0.000,C 180.000} C_DIS
LIN {X 60.964,Y 113.753,Z 66.500,A 180.000,B 0.000,C 180.000} C_DIS
LIN {X 61.500,Y 113.633,Z 66.500,A 180.000,B 0.000,C 180.000} C_DIS
LIN {X 61.679,Y 113.588,Z 66.500,A 180.000,B 0.000,C 180.000} C_DIS
LIN {X 62.215,Y 113.432,Z 66.500,A 180.000,B 0.000,C 180.000} C_DIS
LIN {X 62.394,Y 113.378,Z 66.500,A 180.000,B 0.000,C 180.000} C_DIS
LIN {X 62.491,Y 113.343,Z 66.500,A 180.000,B 0.000,C 180.000} C_DIS
LIN {X 62.987,Y 113.165,Z 66.500,A 180.000,B 0.000,C 180.000} C_DIS
LIN {X 63.109,Y 113.119,Z 66.500,A 180.000,B 0.000,C 180.000} C_DIS
LIN {X 63.288,Y 113.043,Z 66.500,A 180.000,B 0.000,C 180.000} C_DIS
LIN {X 63.645,Y 112.888,Z 66.500,A 180.000,B 0.000,C 180.000} C_DIS
LIN {X 63.824,Y 112.809,Z 66.500,A 180.000,B 0.000,C 180.000} C_DIS
LIN {X 63.829,Y 112.807,Z 66.500,A 180.000,B 0.000,C 180.000} C_DIS
LIN {X 64.003,Y 112.720,Z 66.500,A 180.000,B 0.000,C 180.000} C_DIS
LIN {X 64.360,Y 112.538,Z 66.500,A 180.000,B 0.000,C 180.000} C_DIS
LIN {X 64.530,Y 112.450,Z 66.500,A 180.000,B 0.000,C 180.000} C_DIS
LIN {X 64.539,Y 112.444,Z 66.500,A 180.000,B 0.000,C 180.000} C_DIS
LIN {X 64.718,Y 112.339,Z 66.500,A 180.000,B 0.000,C 180.000} C_DIS
LIN {X 65.075,Y 112.128,Z 66.500,A 180.000,B 0.000,C 180.000} C_DIS
LIN {X 65.136,Y 112.092,Z 66.500,A 180.000,B 0.000,C 180.000} C_DIS
LIN {X 65.254,Y 112.017,Z 66.500,A 180.000,B 0.000,C 180.000} C_DIS
LIN {X 65.433,Y 111.896,Z 66.500,A 180.000,B 0.000,C 180.000} C_DIS
LIN {X 65.670,Y 111.734,Z 66.500,A 180.000,B 0.000,C 180.000} C_DIS
LIN {X 65.791,Y 111.653,Z 66.500,A 180.000,B 0.000,C 180.000} C_DIS
LIN {X 65.923,Y 111.556,Z 66.500,A 180.000,B 0.000,C 180.000} C_DIS
LIN {X 66.384,Y 111.198,Z 66.500,A 180.000,B 0.000,C 180.000} C_DIS
LIN {X 66.506,Y 111.099,Z 66.500,A 180.000,B 0.000,C 180.000} C_DIS
LIN {X 66.597,Y 111.019,Z 66.500,A 180.000,B 0.000,C 180.000} C_DIS
LIN {X 67.002,Y 110.662,Z 66.500,A 180.000,B 0.000,C 180.000} C_DIS
LIN {X 67.042,Y 110.626,Z 66.500,A 180.000,B 0.000,C 180.000} C_DIS
LIN {X 67.188,Y 110.483,Z 66.500,A 180.000,B 0.000,C 180.000} C_DIS
LIN {X 67.545,Y 110.126,Z 66.500,A 180.000,B 0.000,C 180.000} C_DIS
LIN {X 67.578,Y 110.092,Z 66.500,A 180.000,B 0.000,C 180.000} C_DIS
LIN {X 67.711,Y 109.947,Z 66.500,A 180.000,B 0.000,C 180.000} C_DIS
LIN {X 68.026,Y 109.589,Z 66.500,A 180.000,B 0.000,C 180.000} C_DIS
LIN {X 68.115,Y 109.488,Z 66.500,A 180.000,B 0.000,C 180.000} C_DIS
LIN {X 68.177,Y 109.410,Z 66.500,A 180.000,B 0.000,C 180.000} C_DIS
LIN {X 68.472,Y 109.031,Z 66.500,A 180.000,B 0.000,C 180.000} C_DIS
LIN {X 68.593,Y 108.874,Z 66.500,A 180.000,B 0.000,C 180.000} C_DIS
LIN {X 68.651,Y 108.793,Z 66.500,A 180.000,B 0.000,C 180.000} C_DIS
LIN {X 68.717,Y 108.695,Z 66.500,A 180.000,B 0.000,C 180.000} C_DIS
LIN {X 69.008,Y 108.267,Z 66.500,A 180.000,B 0.000,C 180.000} C_DIS
LIN {X 69.078,Y 108.159,Z 66.500,A 180.000,B 0.000,C 180.000} C_DIS
LIN {X 69.184,Y 107.980,Z 66.500,A 180.000,B 0.000,C 180.000} C_DIS
LIN {X 69.396,Y 107.623,Z 66.500,A 180.000,B 0.000,C 180.000} C_DIS
LIN {X 69.495,Y 107.444,Z 66.500,A 180.000,B 0.000,C 180.000} C_DIS
LIN {X 69.768,Y 106.908,Z 66.500,A 180.000,B 0.000,C 180.000} C_DIS
LIN {X 69.852,Y 106.729,Z 66.500,A 180.000,B 0.000,C 180.000} C_DIS
LIN {X 70.084,Y 106.193,Z 66.500,A 180.000,B 0.000,C 180.000} C_DIS
LIN {X 70.155,Y 106.014,Z 66.500,A 180.000,B 0.000,C 180.000} C_DIS
LIN {X 70.348,Y 105.477,Z 66.500,A 180.000,B 0.000,C 180.000} C_DIS
LIN {X 70.408,Y 105.299,Z 66.500,A 180.000,B 0.000,C 180.000} C_DIS
LIN {X 70.439,Y 105.194,Z 66.500,A 180.000,B 0.000,C 180.000} C_DIS
LIN {X 70.564,Y 104.762,Z 66.500,A 180.000,B 0.000,C 180.000} C_DIS
LIN {X 70.614,Y 104.584,Z 66.500,A 180.000,B 0.000,C 180.000} C_DIS
LIN {X 70.617,Y 104.568,Z 66.500,A 180.000,B 0.000,C 180.000} C_DIS
LIN {X 70.654,Y 104.405,Z 66.500,A 180.000,B 0.000,C 180.000} C_DIS
LIN {X 70.734,Y 104.047,Z 66.500,A 180.000,B 0.000,C 180.000} C_DIS
LIN {X 70.773,Y 103.869,Z 66.500,A 180.000,B 0.000,C 180.000} C_DIS
LIN {X 70.796,Y 103.739,Z 66.500,A 180.000,B 0.000,C 180.000} C_DIS
LIN {X 70.889,Y 103.153,Z 66.500,A 180.000,B 0.000,C 180.000} C_DIS
LIN {X 70.911,Y 102.975,Z 66.500,A 180.000,B 0.000,C 180.000} C_DIS
LIN {X 70.962,Y 102.438,Z 66.500,A 180.000,B 0.000,C 180.000} C_DIS
LIN {X 70.975,Y 102.292,Z 66.500,A 180.000,B 0.000,C 180.000} C_DIS
LIN {X 70.977,Y 102.260,Z 66.500,A 180.000,B 0.000,C 180.000} C_DIS
LIN {X 70.983,Y 102.081,Z 66.500,A 180.000,B 0.000,C 180.000} C_DIS
LIN {X 70.994,Y 101.723,Z 66.500,A 180.000,B 0.000,C 180.000} C_DIS
LIN {X 71.000,Y 101.545,Z 66.500,A 180.000,B 0.000,C 180.000} C_DIS
LIN {X 70.997,Y 101.366,Z 66.500,A 180.000,B 0.000,C 180.000} C_DIS
LIN {X 70.980,Y 100.829,Z 66.500,A 180.000,B 0.000,C 180.000} C_DIS
LIN {X 70.975,Y 100.708,Z 66.500,A 180.000,B 0.000,C 180.000} C_DIS
LIN {X 70.970,Y 100.651,Z 66.500,A 180.000,B 0.000,C 180.000} C_DIS
LIN {X 70.954,Y 100.472,Z 66.500,A 180.000,B 0.000,C 180.000} C_DIS
LIN {X 70.920,Y 100.114,Z 66.500,A 180.000,B 0.000,C 180.000} C_DIS
LIN {X 70.902,Y 99.936,Z 66.500,A 180.000,B 0.000,C 180.000} C_DIS
LIN {X 70.875,Y 99.757,Z 66.500,A 180.000,B 0.000,C 180.000} C_DIS
LIN {X 70.796,Y 99.261,Z 66.500,A 180.000,B 0.000,C 180.000} C_DIS
LIN {X 70.790,Y 99.221,Z 66.500,A 180.000,B 0.000,C 180.000} C_DIS
LIN {X 70.754,Y 99.042,Z 66.500,A 180.000,B 0.000,C 180.000} C_DIS
LIN {X 70.670,Y 98.665,Z 66.500,A 180.000,B 0.000,C 180.000} C_DIS
LIN {X 70.634,Y 98.505,Z 66.500,A 180.000,B 0.000,C 180.000} C_DIS
LIN {X 70.617,Y 98.432,Z 66.500,A 180.000,B 0.000,C 180.000} C_DIS
LIN {X 70.590,Y 98.327,Z 66.500,A 180.000,B 0.000,C 180.000} C_DIS
LIN {X 70.538,Y 98.148,Z 66.500,A 180.000,B 0.000,C 180.000} C_DIS
LIN {X 70.434,Y 97.790,Z 66.500,A 180.000,B 0.000,C 180.000} C_DIS
LIN {X 70.380,Y 97.612,Z 66.500,A 180.000,B 0.000,C 180.000} C_DIS
LIN {X 70.316,Y 97.433,Z 66.500,A 180.000,B 0.000,C 180.000} C_DIS
LIN {X 70.187,Y 97.075,Z 66.500,A 180.000,B 0.000,C 180.000} C_DIS
LIN {X 70.121,Y 96.897,Z 66.500,A 180.000,B 0.000,C 180.000} C_DIS
LIN {X 70.081,Y 96.800,Z 66.500,A 180.000,B 0.000,C 180.000} C_DIS
LIN {X 69.891,Y 96.360,Z 66.500,A 180.000,B 0.000,C 180.000} C_DIS
LIN {X 69.812,Y 96.181,Z 66.500,A 180.000,B 0.000,C 180.000} C_DIS
LIN {X 69.724,Y 96.005,Z 66.500,A 180.000,B 0.000,C 180.000} C_DIS
LIN {X 69.540,Y 95.645,Z 66.500,A 180.000,B 0.000,C 180.000} C_DIS
LIN {X 69.447,Y 95.466,Z 66.500,A 180.000,B 0.000,C 180.000} C_DIS
LIN {X 69.366,Y 95.327,Z 66.500,A 180.000,B 0.000,C 180.000} C_DIS
LIN {X 69.131,Y 94.930,Z 66.500,A 180.000,B 0.000,C 180.000} C_DIS
LIN {X 69.021,Y 94.751,Z 66.500,A 180.000,B 0.000,C 180.000} C_DIS
LIN {X 69.008,Y 94.733,Z 66.500,A 180.000,B 0.000,C 180.000} C_DIS
LIN {X 68.657,Y 94.215,Z 66.500,A 180.000,B 0.000,C 180.000} C_DIS
LIN {X 68.651,Y 94.207,Z 66.500,A 180.000,B 0.000,C 180.000} C_DIS
LIN {X 68.524,Y 94.036,Z 66.500,A 180.000,B 0.000,C 180.000} C_DIS
LIN {X 68.247,Y 93.679,Z 66.500,A 180.000,B 0.000,C 180.000} C_DIS
LIN {X 68.115,Y 93.512,Z 66.500,A 180.000,B 0.000,C 180.000} C_DIS
LIN {X 68.104,Y 93.500,Z 66.500,A 180.000,B 0.000,C 180.000} C_DIS
LIN {X 67.947,Y 93.321,Z 66.500,A 180.000,B 0.000,C 180.000} C_DIS
LIN {X 67.757,Y 93.106,Z 66.500,A 180.000,B 0.000,C 180.000} C_DIS
LIN {X 67.631,Y 92.964,Z 66.500,A 180.000,B 0.000,C 180.000} C_DIS
LIN {X 67.578,Y 92.908,Z 66.500,A 180.000,B 0.000,C 180.000} C_DIS
LIN {X 67.456,Y 92.785,Z 66.500,A 180.000,B 0.000,C 180.000} C_DIS
LIN {X 67.221,Y 92.550,Z 66.500,A 180.000,B 0.000,C 180.000} C_DIS
LIN {X 67.098,Y 92.427,Z 66.500,A 180.000,B 0.000,C 180.000} C_DIS
LIN {X 67.042,Y 92.374,Z 66.500,A 180.000,B 0.000,C 180.000} C_DIS
LIN {X 66.901,Y 92.249,Z 66.500,A 180.000,B 0.000,C 180.000} C_DIS
LIN {X 66.684,Y 92.058,Z 66.500,A 180.000,B 0.000,C 180.000} C_DIS
LIN {X 66.506,Y 91.901,Z 66.500,A 180.000,B 0.000,C 180.000} C_DIS
LIN {X 66.494,Y 91.891,Z 66.500,A 180.000,B 0.000,C 180.000} C_DIS
LIN {X 66.327,Y 91.758,Z 66.500,A 180.000,B 0.000,C 180.000} C_DIS
LIN {X 65.969,Y 91.480,Z 66.500,A 180.000,B 0.000,C 180.000} C_DIS
LIN {X 65.801,Y 91.355,Z 66.500,A 180.000,B 0.000,C 180.000} C_DIS
LIN {X 65.791,Y 91.347,Z 66.500,A 180.000,B 0.000,C 180.000} C_DIS
LIN {X 65.538,Y 91.176,Z 66.500,A 180.000,B 0.000,C 180.000} C_DIS
LIN {X 65.275,Y 90.997,Z 66.500,A 180.000,B 0.000,C 180.000} C_DIS
LIN {X 65.254,Y 90.983,Z 66.500,A 180.000,B 0.000,C 180.000} C_DIS
LIN {X 65.075,Y 90.872,Z 66.500,A 180.000,B 0.000,C 180.000} C_DIS
LIN {X 64.682,Y 90.640,Z 66.500,A 180.000,B 0.000,C 180.000} C_DIS
LIN {X 64.539,Y 90.556,Z 66.500,A 180.000,B 0.000,C 180.000} C_DIS
LIN {X 64.360,Y 90.462,Z 66.500,A 180.000,B 0.000,C 180.000} C_DIS
LIN {X 64.003,Y 90.280,Z 66.500,A 180.000,B 0.000,C 180.000} C_DIS
LIN {X 63.824,Y 90.191,Z 66.500,A 180.000,B 0.000,C 180.000} C_DIS
LIN {X 63.645,Y 90.112,Z 66.500,A 180.000,B 0.000,C 180.000} C_DIS
LIN {X 63.213,Y 89.925,Z 66.500,A 180.000,B 0.000,C 180.000} C_DIS
LIN {X 63.109,Y 89.881,Z 66.500,A 180.000,B 0.000,C 180.000} C_DIS
LIN {X 62.930,Y 89.815,Z 66.500,A 180.000,B 0.000,C 180.000} C_DIS
LIN {X 62.573,Y 89.686,Z 66.500,A 180.000,B 0.000,C 180.000} C_DIS
LIN {X 62.394,Y 89.622,Z 66.500,A 180.000,B 0.000,C 180.000} C_DIS
LIN {X 62.215,Y 89.568,Z 66.500,A 180.000,B 0.000,C 180.000} C_DIS
LIN {X 61.679,Y 89.412,Z 66.500,A 180.000,B 0.000,C 180.000} C_DIS
LIN {X 61.591,Y 89.388,Z 66.500,A 180.000,B 0.000,C 180.000} C_DIS
LIN {X 61.500,Y 89.367,Z 66.500,A 180.000,B 0.000,C 180.000} C_DIS
LIN {X 60.964,Y 89.247,Z 66.500,A 180.000,B 0.000,C 180.000} C_DIS
LIN {X 60.785,Y 89.211,Z 66.500,A 180.000,B 0.000,C 180.000} C_DIS
LIN {X 60.774,Y 89.209,Z 66.500,A 180.000,B 0.000,C 180.000} C_DIS
LIN {X 60.606,Y 89.183,Z 66.500,A 180.000,B 0.000,C 180.000} C_DIS
LIN {X 60.249,Y 89.126,Z 66.500,A 180.000,B 0.000,C 180.000} C_DIS
LIN {X 60.070,Y 89.099,Z 66.500,A 180.000,B 0.000,C 180.000} C_DIS
LIN {X 59.891,Y 89.081,Z 66.500,A 180.000,B 0.000,C 180.000} C_DIS
LIN {X 59.361,Y 89.031,Z 66.500,A 180.000,B 0.000,C 180.000} C_DIS
LIN {X 59.355,Y 89.030,Z 66.500,A 180.000,B 0.000,C 180.000} C_DIS
LIN {X 59.176,Y 89.020,Z 66.500,A 180.000,B 0.000,C 180.000} C_DIS
LIN {X 58.640,Y 89.003,Z 66.500,A 180.000,B 0.000,C 180.000} C_DIS
LIN {X 58.461,Y 89.000,Z 66.500,A 180.000,B 0.000,C 180.000} C_DIS
LIN {X 58.282,Y 89.006,Z 66.500,A 180.000,B 0.000,C 180.000} C_DIS
LIN {X 57.925,Y 89.017,Z 66.500,A 180.000,B 0.000,C 180.000} C_DIS
LIN {X 57.746,Y 89.023,Z 66.500,A 180.000,B 0.000,C 180.000} C_DIS
LIN {X 57.639,Y 89.031,Z 66.500,A 180.000,B 0.000,C 180.000} C_DIS
LIN {X 57.031,Y 89.088,Z 66.500,A 180.000,B 0.000,C 180.000} C_DIS
LIN {X 56.852,Y 89.110,Z 66.500,A 180.000,B 0.000,C 180.000} C_DIS
LIN {X 56.316,Y 89.195,Z 66.500,A 180.000,B 0.000,C 180.000} C_DIS
LIN {X 56.226,Y 89.209,Z 66.500,A 180.000,B 0.000,C 180.000} C_DIS
LIN {X 56.137,Y 89.225,Z 66.500,A 180.000,B 0.000,C 180.000} C_DIS
LIN {X 55.958,Y 89.265,Z 66.500,A 180.000,B 0.000,C 180.000} C_DIS
LIN {X 55.601,Y 89.345,Z 66.500,A 180.000,B 0.000,C 180.000} C_DIS
LIN {X 55.422,Y 89.385,Z 66.500,A 180.000,B 0.000,C 180.000} C_DIS
LIN {X 55.409,Y 89.388,Z 66.500,A 180.000,B 0.000,C 180.000} C_DIS
LIN {X 55.243,Y 89.434,Z 66.500,A 180.000,B 0.000,C 180.000} C_DIS
LIN {X 54.787,Y 89.567,Z 66.500,A 180.000,B 0.000,C 180.000} C_DIS
LIN {X 54.707,Y 89.590,Z 66.500,A 180.000,B 0.000,C 180.000} C_DIS
LIN {X 54.528,Y 89.650,Z 66.500,A 180.000,B 0.000,C 180.000} C_DIS
LIN {X 53.992,Y 89.843,Z 66.500,A 180.000,B 0.000,C 180.000} C_DIS
LIN {X 53.813,Y 89.913,Z 66.500,A 180.000,B 0.000,C 180.000} C_DIS
LIN {X 53.277,Y 90.146,Z 66.500,A 180.000,B 0.000,C 180.000} C_DIS
LIN {X 53.098,Y 90.229,Z 66.500,A 180.000,B 0.000,C 180.000} C_DIS
LIN {X 52.562,Y 90.502,Z 66.500,A 180.000,B 0.000,C 180.000} C_DIS
LIN {X 52.383,Y 90.601,Z 66.500,A 180.000,B 0.000,C 180.000} C_DIS
LIN {X 52.015,Y 90.818,Z 66.500,A 180.000,B 0.000,C 180.000} C_DIS
LIN {X 51.847,Y 90.918,Z 66.500,A 180.000,B 0.000,C 180.000} C_DIS
LIN {X 51.725,Y 90.997,Z 66.500,A 180.000,B 0.000,C 180.000} C_DIS
LIN {X 51.310,Y 91.279,Z 66.500,A 180.000,B 0.000,C 180.000} C_DIS
LIN {X 51.199,Y 91.355,Z 66.500,A 180.000,B 0.000,C 180.000} C_DIS
LIN {X 51.131,Y 91.403,Z 66.500,A 180.000,B 0.000,C 180.000} C_DIS
LIN {X 50.962,Y 91.533,Z 66.500,A 180.000,B 0.000,C 180.000} C_DIS
LIN {X 50.595,Y 91.818,Z 66.500,A 180.000,B 0.000,C 180.000} C_DIS
LIN {X 50.506,Y 91.891,Z 66.500,A 180.000,B 0.000,C 180.000} C_DIS
LIN {X 50.416,Y 91.969,Z 66.500,A 180.000,B 0.000,C 180.000} C_DIS
LIN {X 50.059,Y 92.284,Z 66.500,A 180.000,B 0.000,C 180.000} C_DIS
LIN {X 49.902,Y 92.427,Z 66.500,A 180.000,B 0.000,C 180.000} C_DIS
LIN {X 49.880,Y 92.449,Z 66.500,A 180.000,B 0.000,C 180.000} C_DIS
LIN {X 49.523,Y 92.807,Z 66.500,A 180.000,B 0.000,C 180.000} C_DIS
LIN {X 49.369,Y 92.964,Z 66.500,A 180.000,B 0.000,C 180.000} C_DIS
LIN {X 49.344,Y 92.991,Z 66.500,A 180.000,B 0.000,C 180.000} C_DIS
LIN {X 49.211,Y 93.142,Z 66.500,A 180.000,B 0.000,C 180.000} C_DIS
LIN {X 48.986,Y 93.397,Z 66.500,A 180.000,B 0.000,C 180.000} C_DIS
LIN {X 48.896,Y 93.500,Z 66.500,A 180.000,B 0.000,C 180.000} C_DIS
LIN {X 48.807,Y 93.609,Z 66.500,A 180.000,B 0.000,C 180.000} C_DIS
LIN {X 48.450,Y 94.070,Z 66.500,A 180.000,B 0.000,C 180.000} C_DIS
LIN {X 48.343,Y 94.215,Z 66.500,A 180.000,B 0.000,C 180.000} C_DIS
LIN {X 48.092,Y 94.584,Z 66.500,A 180.000,B 0.000,C 180.000} C_DIS
LIN {X 47.979,Y 94.751,Z 66.500,A 180.000,B 0.000,C 180.000} C_DIS
LIN {X 47.914,Y 94.855,Z 66.500,A 180.000,B 0.000,C 180.000} C_DIS
LIN {X 47.869,Y 94.930,Z 66.500,A 180.000,B 0.000,C 180.000} C_DIS
LIN {X 47.657,Y 95.288,Z 66.500,A 180.000,B 0.000,C 180.000} C_DIS
LIN {X 47.556,Y 95.460,Z 66.500,A 180.000,B 0.000,C 180.000} C_DIS
LIN {X 47.553,Y 95.466,Z 66.500,A 180.000,B 0.000,C 180.000} C_DIS
LIN {X 47.460,Y 95.645,Z 66.500,A 180.000,B 0.000,C 180.000} C_DIS
LIN {X 47.277,Y 96.003,Z 66.500,A 180.000,B 0.000,C 180.000} C_DIS
LIN {X 47.198,Y 96.159,Z 66.500,A 180.000,B 0.000,C 180.000} C_DIS
LIN {X 47.188,Y 96.181,Z 66.500,A 180.000,B 0.000,C 180.000} C_DIS
LIN {X 47.109,Y 96.360,Z 66.500,A 180.000,B 0.000,C 180.000} C_DIS
LIN {X 46.955,Y 96.718,Z 66.500,A 180.000,B 0.000,C 180.000} C_DIS
LIN {X 46.879,Y 96.897,Z 66.500,A 180.000,B 0.000,C 180.000} C_DIS
LIN {X 46.841,Y 96.997,Z 66.500,A 180.000,B 0.000,C 180.000} C_DIS
LIN {X 46.662,Y 97.494,Z 66.500,A 180.000,B 0.000,C 180.000} C_DIS
LIN {X 46.620,Y 97.612,Z 66.500,A 180.000,B 0.000,C 180.000} C_DIS
LIN {X 46.566,Y 97.790,Z 66.500,A 180.000,B 0.000,C 180.000} C_DIS
LIN {X 46.462,Y 98.148,Z 66.500,A 180.000,B 0.000,C 180.000} C_DIS
LIN {X 46.410,Y 98.327,Z 66.500,A 180.000,B 0.000,C 180.000} C_DIS
LIN {X 46.366,Y 98.505,Z 66.500,A 180.000,B 0.000,C 180.000} C_DIS
LIN {X 46.246,Y 99.042,Z 66.500,A 180.000,B 0.000,C 180.000} C_DIS
LIN {X 46.210,Y 99.221,Z 66.500,A 180.000,B 0.000,C 180.000} C_DIS
LIN {X 46.182,Y 99.399,Z 66.500,A 180.000,B 0.000,C 180.000} C_DIS
LIN {X 46.126,Y 99.753,Z 66.500,A 180.000,B 0.000,C 180.000} C_DIS
LIN {X 46.125,Y 99.757,Z 66.500,A 180.000,B 0.000,C 180.000} C_DIS
LIN {X 46.098,Y 99.936,Z 66.500,A 180.000,B 0.000,C 180.000} C_DIS
LIN {X 46.080,Y 100.114,Z 66.500,A 180.000,B 0.000,C 180.000} C_DIS
LIN {X 46.046,Y 100.472,Z 66.500,A 180.000,B 0.000,C 180.000} C_DIS
LIN {X 46.030,Y 100.651,Z 66.500,A 180.000,B 0.000,C 180.000} C_DIS
LIN {X 46.020,Y 100.829,Z 66.500,A 180.000,B 0.000,C 180.000} C_DIS
LIN {X 46.003,Y 101.366,Z 66.500,A 180.000,B 0.000,C 180.000} C_DIS
LIN {X 46.000,Y 101.545,Z 66.500,A 180.000,B 0.000,C 180.000} C_DIS
LIN {X 46.006,Y 101.723,Z 66.500,A 180.000,B 0.000,C 180.000} C_DIS
LIN {X 46.017,Y 102.081,Z 66.500,A 180.000,B 0.000,C 180.000} C_DIS
LIN {X 46.023,Y 102.260,Z 66.500,A 180.000,B 0.000,C 180.000} C_DIS
LIN {X 46.038,Y 102.438,Z 66.500,A 180.000,B 0.000,C 180.000} C_DIS
LIN {X 46.089,Y 102.975,Z 66.500,A 180.000,B 0.000,C 180.000} C_DIS
LIN {X 46.111,Y 103.153,Z 66.500,A 180.000,B 0.000,C 180.000} C_DIS
LIN {X 46.196,Y 103.690,Z 66.500,A 180.000,B 0.000,C 180.000} C_DIS
LIN {X 46.227,Y 103.869,Z 66.500,A 180.000,B 0.000,C 180.000} C_DIS
LIN {X 46.266,Y 104.047,Z 66.500,A 180.000,B 0.000,C 180.000} C_DIS
LIN {X 46.346,Y 104.405,Z 66.500,A 180.000,B 0.000,C 180.000} C_DIS
LIN {X 46.386,Y 104.584,Z 66.500,A 180.000,B 0.000,C 180.000} C_DIS
LIN {X 46.436,Y 104.762,Z 66.500,A 180.000,B 0.000,C 180.000} C_DIS
LIN {X 46.540,Y 105.120,Z 66.500,A 180.000,B 0.000,C 180.000} C_DIS
LIN {X 46.592,Y 105.299,Z 66.500,A 180.000,B 0.000,C 180.000} C_DIS
LIN {X 46.652,Y 105.477,Z 66.500,A 180.000,B 0.000,C 180.000} C_DIS
LIN {X 46.845,Y 106.014,Z 66.500,A 180.000,B 0.000,C 180.000} C_DIS
LIN {X 46.916,Y 106.193,Z 66.500,A 180.000,B 0.000,C 180.000} C_DIS
LIN {X 47.148,Y 106.729,Z 66.500,A 180.000,B 0.000,C 180.000} C_DIS
LIN {X 47.198,Y 106.841,Z 66.500,A 180.000,B 0.000,C 180.000} C_DIS
LIN {X 47.232,Y 106.908,Z 66.500,A 180.000,B 0.000,C 180.000} C_DIS
LIN {X 47.505,Y 107.444,Z 66.500,A 180.000,B 0.000,C 180.000} C_DIS
LIN {X 47.556,Y 107.540,Z 66.500,A 180.000,B 0.000,C 180.000} C_DIS
LIN {X 47.604,Y 107.623,Z 66.500,A 180.000,B 0.000,C 180.000} C_DIS
LIN {X 47.816,Y 107.980,Z 66.500,A 180.000,B 0.000,C 180.000} C_DIS
LIN {X 47.914,Y 108.145,Z 66.500,A 180.000,B 0.000,C 180.000} C_DIS
LIN {X 47.922,Y 108.159,Z 66.500,A 180.000,B 0.000,C 180.000} C_DIS
LIN {X 48.040,Y 108.338,Z 66.500,A 180.000,B 0.000,C 180.000} C_DIS
LIN {X 48.283,Y 108.695,Z 66.500,A 180.000,B 0.000,C 180.000} C_DIS
LIN {X 48.407,Y 108.874,Z 66.500,A 180.000,B 0.000,C 180.000} C_DIS
LIN {X 48.450,Y 108.930,Z 66.500,A 180.000,B 0.000,C 180.000} C_DIS
LIN {X 48.823,Y 109.410,Z 66.500,A 180.000,B 0.000,C 180.000} C_DIS
LIN {X 48.974,Y 109.589,Z 66.500,A 180.000,B 0.000,C 180.000} C_DIS
LIN {X 49.289,Y 109.947,Z 66.500,A 180.000,B 0.000,C 180.000} C_DIS
LIN {X 49.344,Y 110.009,Z 66.500,A 180.000,B 0.000,C 180.000} C_DIS
LIN {X 49.455,Y 110.126,Z 66.500,A 180.000,B 0.000,C 180.000} C_DIS
LIN {X 49.880,Y 110.551,Z 66.500,A 180.000,B 0.000,C 180.000} C_DIS
LIN {X 49.998,Y 110.662,Z 66.500,A 180.000,B 0.000,C 180.000} C_DIS
LIN {X 50.416,Y 111.031,Z 66.500,A 180.000,B 0.000,C 180.000} C_DIS
LIN {X 50.595,Y 111.182,Z 66.500,A 180.000,B 0.000,C 180.000} C_DIS
LIN {X 51.077,Y 111.556,Z 66.500,A 180.000,B 0.000,C 180.000} C_DIS
LIN {X 51.131,Y 111.597,Z 66.500,A 180.000,B 0.000,C 180.000} C_DIS
LIN {X 51.310,Y 111.721,Z 66.500,A 180.000,B 0.000,C 180.000} C_DIS
LIN {X 51.668,Y 111.964,Z 66.500,A 180.000,B 0.000,C 180.000} C_DIS
LIN {X 51.847,Y 112.082,Z 66.500,A 180.000,B 0.000,C 180.000} C_DIS
LIN {X 51.864,Y 112.092,Z 66.500,A 180.000,B 0.000,C 180.000} C_DIS
LIN {X 52.204,Y 112.293,Z 66.500,A 180.000,B 0.000,C 180.000} C_DIS
LIN {X 52.383,Y 112.399,Z 66.500,A 180.000,B 0.000,C 180.000} C_DIS
LIN {X 52.470,Y 112.450,Z 66.500,A 180.000,B 0.000,C 180.000} C_DIS
LIN {X 52.562,Y 112.498,Z 66.500,A 180.000,B 0.000,C 180.000} C_DIS
LIN {X 53.098,Y 112.771,Z 66.500,A 180.000,B 0.000,C 180.000} C_DIS
LIN {X 53.171,Y 112.807,Z 66.500,A 180.000,B 0.000,C 180.000} C_DIS
LIN {X 53.277,Y 112.854,Z 66.500,A 180.000,B 0.000,C 180.000} C_DIS
LIN {X 53.813,Y 113.087,Z 66.500,A 180.000,B 0.000,C 180.000} C_DIS
LIN {X 53.992,Y 113.157,Z 66.500,A 180.000,B 0.000,C 180.000} C_DIS
LIN {X 54.528,Y 113.350,Z 66.500,A 180.000,B 0.000,C 180.000} C_DIS
LIN {X 54.707,Y 113.410,Z 66.500,A 180.000,B 0.000,C 180.000} C_DIS
LIN {X 55.243,Y 113.566,Z 66.500,A 180.000,B 0.000,C 180.000} C_DIS
LIN {X 55.422,Y 113.615,Z 66.500,A 180.000,B 0.000,C 180.000} C_DIS
LIN {X 55.601,Y 113.655,Z 66.500,A 180.000,B 0.000,C 180.000} C_DIS
LIN {X 55.958,Y 113.735,Z 66.500,A 180.000,B 0.000,C 180.000} C_DIS
LIN {X 56.066,Y 113.759,Z 66.500,A 180.000,B 0.000,C 180.000} C_DIS
; Link Move Starts
LIN {X 56.207,Y 113.838,Z 66.500,A 180.000,B 0.000,C 180.000} C_DIS
LIN {X 56.366,Y 113.863,Z 66.500,A 180.000,B 0.000,C 180.000} C_DIS
LIN {X 56.677,Y 113.913,Z 66.499,A 180.000,B 0.000,C 180.000} C_DIS
LIN {X 56.989,Y 113.958,Z 66.498,A 180.000,B 0.000,C 180.000} C_DIS
LIN {X 57.302,Y 113.988,Z 66.496,A 180.000,B 0.000,C 180.000} C_DIS
LIN {X 57.616,Y 114.017,Z 66.494,A 180.000,B 0.000,C 180.000} C_DIS
LIN {X 57.930,Y 114.033,Z 66.491,A 180.000,B 0.000,C 180.000} C_DIS
LIN {X 58.245,Y 114.043,Z 66.488,A 180.000,B 0.000,C 180.000} C_DIS
LIN {X 58.560,Y 114.049,Z 66.485,A 180.000,B 0.000,C 180.000} C_DIS
LIN {X 58.875,Y 114.039,Z 66.481,A 180.000,B 0.000,C 180.000} C_DIS
LIN {X 59.190,Y 114.030,Z 66.477,A 180.000,B 0.000,C 180.000} C_DIS
LIN {X 59.504,Y 114.006,Z 66.472,A 180.000,B 0.000,C 180.000} C_DIS
LIN {X 59.661,Y 113.991,Z 66.470,A 180.000,B 0.000,C 180.000} C_DIS
LIN {X 59.817,Y 113.976,Z 66.467,A 180.000,B 0.000,C 180.000} C_DIS
LIN {X 59.974,Y 113.962,Z 66.464,A 180.000,B 0.000,C 180.000} C_DIS
LIN {X 60.131,Y 113.943,Z 66.462,A 180.000,B 0.000,C 180.000} C_DIS
LIN {X 60.286,Y 113.919,Z 66.459,A 180.000,B 0.000,C 180.000} C_DIS
LIN {X 60.442,Y 113.894,Z 66.456,A 180.000,B 0.000,C 180.000} C_DIS
LIN {X 60.597,Y 113.869,Z 66.453,A 180.000,B 0.000,C 180.000} C_DIS
LIN {X 60.753,Y 113.845,Z 66.450,A 180.000,B 0.000,C 180.000} C_DIS
LIN {X 60.908,Y 113.816,Z 66.446,A 180.000,B 0.000,C 180.000} C_DIS
LIN {X 61.062,Y 113.782,Z 66.443,A 180.000,B 0.000,C 180.000} C_DIS
LIN {X 61.215,Y 113.748,Z 66.440,A 180.000,B 0.000,C 180.000} C_DIS
LIN {X 61.369,Y 113.713,Z 66.436,A 180.000,B 0.000,C 180.000} C_DIS
LIN {X 61.523,Y 113.679,Z 66.433,A 180.000,B 0.000,C 180.000} C_DIS
LIN {X 61.676,Y 113.641,Z 66.429,A 180.000,B 0.000,C 180.000} C_DIS
LIN {X 61.827,Y 113.597,Z 66.425,A 180.000,B 0.000,C 180.000} C_DIS
LIN {X 61.978,Y 113.553,Z 66.421,A 180.000,B 0.000,C 180.000} C_DIS
LIN {X 62.129,Y 113.509,Z 66.417,A 180.000,B 0.000,C 180.000} C_DIS
LIN {X 62.281,Y 113.465,Z 66.413,A 180.000,B 0.000,C 180.000} C_DIS
LIN {X 62.431,Y 113.418,Z 66.409,A 180.000,B 0.000,C 180.000} C_DIS
LIN {X 62.579,Y 113.365,Z 66.405,A 180.000,B 0.000,C 180.000} C_DIS
LIN {X 62.727,Y 113.311,Z 66.401,A 180.000,B 0.000,C 180.000} C_DIS
LIN {X 62.875,Y 113.258,Z 66.397,A 180.000,B 0.000,C 180.000} C_DIS
LIN {X 63.024,Y 113.205,Z 66.392,A 180.000,B 0.000,C 180.000} C_DIS
LIN {X 63.171,Y 113.148,Z 66.388,A 180.000,B 0.000,C 180.000} C_DIS
LIN {X 63.315,Y 113.086,Z 66.383,A 180.000,B 0.000,C 180.000} C_DIS
LIN {X 63.460,Y 113.023,Z 66.379,A 180.000,B 0.000,C 180.000} C_DIS
LIN {X 63.604,Y 112.960,Z 66.374,A 180.000,B 0.000,C 180.000} C_DIS
LIN {X 63.749,Y 112.898,Z 66.369,A 180.000,B 0.000,C 180.000} C_DIS
LIN {X 63.892,Y 112.832,Z 66.365,A 180.000,B 0.000,C 180.000} C_DIS
LIN {X 64.032,Y 112.761,Z 66.360,A 180.000,B 0.000,C 180.000} C_DIS
LIN {X 64.173,Y 112.689,Z 66.355,A 180.000,B 0.000,C 180.000} C_DIS
LIN {X 64.243,Y 112.654,Z 66.352,A 180.000,B 0.000,C 180.000} C_DIS
LIN {X 64.383,Y 112.582,Z 66.347,A 180.000,B 0.000,C 180.000} C_DIS
LIN {X 64.453,Y 112.546,Z 66.345,A 180.000,B 0.000,C 180.000} C_DIS
LIN {X 64.523,Y 112.510,Z 66.342,A 180.000,B 0.000,C 180.000} C_DIS
LIN {X 64.592,Y 112.472,Z 66.340,A 180.000,B 0.000,C 180.000} C_DIS
LIN {X 64.660,Y 112.432,Z 66.337,A 180.000,B 0.000,C 180.000} C_DIS
LIN {X 64.795,Y 112.352,Z 66.332,A 180.000,B 0.000,C 180.000} C_DIS
LIN {X 64.863,Y 112.312,Z 66.329,A 180.000,B 0.000,C 180.000} C_DIS
LIN {X 64.999,Y 112.231,Z 66.324,A 180.000,B 0.000,C 180.000} C_DIS
LIN {X 65.134,Y 112.151,Z 66.319,A 180.000,B 0.000,C 180.000} C_DIS
LIN {X 65.202,Y 112.111,Z 66.316,A 180.000,B 0.000,C 180.000} C_DIS
LIN {X 65.268,Y 112.068,Z 66.313,A 180.000,B 0.000,C 180.000} C_DIS
LIN {X 65.333,Y 112.024,Z 66.310,A 180.000,B 0.000,C 180.000} C_DIS
LIN {X 65.529,Y 111.891,Z 66.302,A 180.000,B 0.000,C 180.000} C_DIS
LIN {X 65.724,Y 111.758,Z 66.294,A 180.000,B 0.000,C 180.000} C_DIS
LIN {X 65.789,Y 111.714,Z 66.291,A 180.000,B 0.000,C 180.000} C_DIS
LIN {X 65.854,Y 111.669,Z 66.288,A 180.000,B 0.000,C 180.000} C_DIS
LIN {X 65.918,Y 111.623,Z 66.286,A 180.000,B 0.000,C 180.000} C_DIS
LIN {X 65.980,Y 111.575,Z 66.283,A 180.000,B 0.000,C 180.000} C_DIS
LIN {X 66.104,Y 111.478,Z 66.277,A 180.000,B 0.000,C 180.000} C_DIS
LIN {X 66.167,Y 111.430,Z 66.275,A 180.000,B 0.000,C 180.000} C_DIS
LIN {X 66.291,Y 111.333,Z 66.269,A 180.000,B 0.000,C 180.000} C_DIS
LIN {X 66.416,Y 111.237,Z 66.264,A 180.000,B 0.000,C 180.000} C_DIS
LIN {X 66.477,Y 111.188,Z 66.261,A 180.000,B 0.000,C 180.000} C_DIS
LIN {X 66.538,Y 111.138,Z 66.258,A 180.000,B 0.000,C 180.000} C_DIS
LIN {X 66.597,Y 111.086,Z 66.256,A 180.000,B 0.000,C 180.000} C_DIS
LIN {X 66.656,Y 111.034,Z 66.253,A 180.000,B 0.000,C 180.000} C_DIS
LIN {X 66.774,Y 110.929,Z 66.247,A 180.000,B 0.000,C 180.000} C_DIS
LIN {X 66.952,Y 110.773,Z 66.239,A 180.000,B 0.000,C 180.000} C_DIS
LIN {X 67.011,Y 110.721,Z 66.236,A 180.000,B 0.000,C 180.000} C_DIS
LIN {X 67.069,Y 110.669,Z 66.233,A 180.000,B 0.000,C 180.000} C_DIS
LIN {X 67.127,Y 110.615,Z 66.231,A 180.000,B 0.000,C 180.000} C_DIS
LIN {X 67.182,Y 110.559,Z 66.228,A 180.000,B 0.000,C 180.000} C_DIS
LIN {X 67.294,Y 110.448,Z 66.222,A 180.000,B 0.000,C 180.000} C_DIS
LIN {X 67.349,Y 110.392,Z 66.220,A 180.000,B 0.000,C 180.000} C_DIS
LIN {X 67.461,Y 110.281,Z 66.214,A 180.000,B 0.000,C 180.000} C_DIS
LIN {X 67.572,Y 110.169,Z 66.209,A 180.000,B 0.000,C 180.000} C_DIS
LIN {X 67.628,Y 110.113,Z 66.206,A 180.000,B 0.000,C 180.000} C_DIS
LIN {X 67.681,Y 110.056,Z 66.203,A 180.000,B 0.000,C 180.000} C_DIS
LIN {X 67.733,Y 109.997,Z 66.201,A 180.000,B 0.000,C 180.000} C_DIS
LIN {X 67.786,Y 109.938,Z 66.198,A 180.000,B 0.000,C 180.000} C_DIS
LIN {X 67.890,Y 109.819,Z 66.192,A 180.000,B 0.000,C 180.000} C_DIS
LIN {X 68.098,Y 109.583,Z 66.181,A 180.000,B 0.000,C 180.000} C_DIS
LIN {X 68.150,Y 109.524,Z 66.178,A 180.000,B 0.000,C 180.000} C_DIS
LIN {X 68.200,Y 109.463,Z 66.176,A 180.000,B 0.000,C 180.000} C_DIS
LIN {X 68.248,Y 109.401,Z 66.173,A 180.000,B 0.000,C 180.000} C_DIS
LIN {X 68.345,Y 109.276,Z 66.167,A 180.000,B 0.000,C 180.000} C_DIS
LIN {X 68.441,Y 109.152,Z 66.162,A 180.000,B 0.000,C 180.000} C_DIS
LIN {X 68.586,Y 108.965,Z 66.154,A 180.000,B 0.000,C 180.000} C_DIS
LIN {X 68.634,Y 108.903,Z 66.151,A 180.000,B 0.000,C 180.000} C_DIS
LIN {X 68.680,Y 108.839,Z 66.148,A 180.000,B 0.000,C 180.000} C_DIS
LIN {X 68.725,Y 108.774,Z 66.145,A 180.000,B 0.000,C 180.000} C_DIS
LIN {X 68.813,Y 108.644,Z 66.140,A 180.000,B 0.000,C 180.000} C_DIS
LIN {X 69.034,Y 108.318,Z 66.126,A 180.000,B 0.000,C 180.000} C_DIS
LIN {X 69.078,Y 108.253,Z 66.123,A 180.000,B 0.000,C 180.000} C_DIS
LIN {X 69.120,Y 108.186,Z 66.121,A 180.000,B 0.000,C 180.000} C_DIS
LIN {X 69.161,Y 108.118,Z 66.118,A 180.000,B 0.000,C 180.000} C_DIS
LIN {X 69.401,Y 107.712,Z 66.101,A 180.000,B 0.000,C 180.000} C_DIS
LIN {X 69.441,Y 107.644,Z 66.099,A 180.000,B 0.000,C 180.000} C_DIS
LIN {X 69.481,Y 107.576,Z 66.096,A 180.000,B 0.000,C 180.000} C_DIS
LIN {X 69.519,Y 107.507,Z 66.093,A 180.000,B 0.000,C 180.000} C_DIS
LIN {X 69.555,Y 107.437,Z 66.090,A 180.000,B 0.000,C 180.000} C_DIS
LIN {X 69.734,Y 107.086,Z 66.077,A 180.000,B 0.000,C 180.000} C_DIS
LIN {X 69.805,Y 106.945,Z 66.071,A 180.000,B 0.000,C 180.000} C_DIS
LIN {X 69.840,Y 106.875,Z 66.068,A 180.000,B 0.000,C 180.000} C_DIS
LIN {X 69.874,Y 106.804,Z 66.066,A 180.000,B 0.000,C 180.000} C_DIS
LIN {X 69.905,Y 106.732,Z 66.063,A 180.000,B 0.000,C 180.000} C_DIS
LIN {X 70.124,Y 106.226,Z 66.044,A 180.000,B 0.000,C 180.000} C_DIS
LIN {X 70.155,Y 106.153,Z 66.041,A 180.000,B 0.000,C 180.000} C_DIS
LIN {X 70.184,Y 106.080,Z 66.038,A 180.000,B 0.000,C 180.000} C_DIS
LIN {X 70.211,Y 106.006,Z 66.035,A 180.000,B 0.000,C 180.000} C_DIS
LIN {X 70.398,Y 105.487,Z 66.016,A 180.000,B 0.000,C 180.000} C_DIS
LIN {X 70.424,Y 105.413,Z 66.013,A 180.000,B 0.000,C 180.000} C_DIS
LIN {X 70.448,Y 105.338,Z 66.011,A 180.000,B 0.000,C 180.000} C_DIS
LIN {X 70.471,Y 105.263,Z 66.008,A 180.000,B 0.000,C 180.000} C_DIS
LIN {X 70.624,Y 104.733,Z 65.989,A 180.000,B 0.000,C 180.000} C_DIS
LIN {X 70.646,Y 104.658,Z 65.986,A 180.000,B 0.000,C 180.000} C_DIS
LIN {X 70.666,Y 104.581,Z 65.983,A 180.000,B 0.000,C 180.000} C_DIS
LIN {X 70.683,Y 104.505,Z 65.980,A 180.000,B 0.000,C 180.000} C_DIS
LIN {X 70.803,Y 103.967,Z 65.961,A 180.000,B 0.000,C 180.000} C_DIS
LIN {X 70.820,Y 103.890,Z 65.959,A 180.000,B 0.000,C 180.000} C_DIS
LIN {X 70.835,Y 103.812,Z 65.956,A 180.000,B 0.000,C 180.000} C_DIS
LIN {X 70.848,Y 103.735,Z 65.953,A 180.000,B 0.000,C 180.000} C_DIS
LIN {X 70.934,Y 103.190,Z 65.934,A 180.000,B 0.000,C 180.000} C_DIS
LIN {X 70.946,Y 103.112,Z 65.931,A 180.000,B 0.000,C 180.000} C_DIS
LIN {X 70.956,Y 103.034,Z 65.928,A 180.000,B 0.000,C 180.000} C_DIS
LIN {X 70.963,Y 102.956,Z 65.926,A 180.000,B 0.000,C 180.000} C_DIS
LIN {X 71.000,Y 102.564,Z 65.912,A 180.000,B 0.000,C 180.000} C_DIS
LIN {X 71.015,Y 102.407,Z 65.906,A 180.000,B 0.000,C 180.000} C_DIS
LIN {X 71.022,Y 102.328,Z 65.904,A 180.000,B 0.000,C 180.000} C_DIS
LIN {X 71.027,Y 102.250,Z 65.901,A 180.000,B 0.000,C 180.000} C_DIS
LIN {X 71.030,Y 102.171,Z 65.898,A 180.000,B 0.000,C 180.000} C_DIS
LIN {X 71.047,Y 101.620,Z 65.879,A 180.000,B 0.000,C 180.000} C_DIS
LIN {X 71.050,Y 101.541,Z 65.876,A 180.000,B 0.000,C 180.000} C_DIS
LIN {X 71.050,Y 101.463,Z 65.873,A 180.000,B 0.000,C 180.000} C_DIS
LIN {X 71.048,Y 101.384,Z 65.871,A 180.000,B 0.000,C 180.000} C_DIS
LIN {X 71.043,Y 101.227,Z 65.865,A 180.000,B 0.000,C 180.000} C_DIS
LIN {X 71.030,Y 100.833,Z 65.851,A 180.000,B 0.000,C 180.000} C_DIS
LIN {X 71.028,Y 100.754,Z 65.849,A 180.000,B 0.000,C 180.000} C_DIS
LIN {X 71.023,Y 100.676,Z 65.846,A 180.000,B 0.000,C 180.000} C_DIS
LIN {X 71.016,Y 100.597,Z 65.843,A 180.000,B 0.000,C 180.000} C_DIS
LIN {X 70.971,Y 100.127,Z 65.827,A 180.000,B 0.000,C 180.000} C_DIS
LIN {X 70.964,Y 100.048,Z 65.824,A 180.000,B 0.000,C 180.000} C_DIS
LIN {X 70.956,Y 99.970,Z 65.821,A 180.000,B 0.000,C 180.000} C_DIS
LIN {X 70.946,Y 99.892,Z 65.818,A 180.000,B 0.000,C 180.000} C_DIS
LIN {X 70.934,Y 99.814,Z 65.816,A 180.000,B 0.000,C 180.000} C_DIS
LIN {X 70.922,Y 99.736,Z 65.813,A 180.000,B 0.000,C 180.000} C_DIS
LIN {X 70.897,Y 99.581,Z 65.807,A 180.000,B 0.000,C 180.000} C_DIS
LIN {X 70.848,Y 99.270,Z 65.796,A 180.000,B 0.000,C 180.000} C_DIS
LIN {X 70.836,Y 99.192,Z 65.794,A 180.000,B 0.000,C 180.000} C_DIS
LIN {X 70.821,Y 99.114,Z 65.791,A 180.000,B 0.000,C 180.000} C_DIS
LIN {X 70.804,Y 99.038,Z 65.788,A 180.000,B 0.000,C 180.000} C_DIS
LIN {X 70.770,Y 98.884,Z 65.783,A 180.000,B 0.000,C 180.000} C_DIS
LIN {X 70.753,Y 98.807,Z 65.780,A 180.000,B 0.000,C 180.000} C_DIS
LIN {X 70.718,Y 98.653,Z 65.774,A 180.000,B 0.000,C 180.000} C_DIS
LIN {X 70.684,Y 98.500,Z 65.769,A 180.000,B 0.000,C 180.000} C_DIS
LIN {X 70.667,Y 98.423,Z 65.766,A 180.000,B 0.000,C 180.000} C_DIS
LIN {X 70.647,Y 98.346,Z 65.763,A 180.000,B 0.000,C 180.000} C_DIS
LIN {X 70.626,Y 98.271,Z 65.761,A 180.000,B 0.000,C 180.000} C_DIS
LIN {X 70.604,Y 98.195,Z 65.758,A 180.000,B 0.000,C 180.000} C_DIS
LIN {X 70.560,Y 98.044,Z 65.752,A 180.000,B 0.000,C 180.000} C_DIS
LIN {X 70.494,Y 97.817,Z 65.744,A 180.000,B 0.000,C 180.000} C_DIS
LIN {X 70.472,Y 97.741,Z 65.741,A 180.000,B 0.000,C 180.000} C_DIS
LIN {X 70.450,Y 97.666,Z 65.739,A 180.000,B 0.000,C 180.000} C_DIS
LIN {X 70.425,Y 97.591,Z 65.736,A 180.000,B 0.000,C 180.000} C_DIS
LIN {X 70.399,Y 97.517,Z 65.733,A 180.000,B 0.000,C 180.000} C_DIS
LIN {X 70.346,Y 97.368,Z 65.728,A 180.000,B 0.000,C 180.000} C_DIS
LIN {X 70.319,Y 97.294,Z 65.725,A 180.000,B 0.000,C 180.000} C_DIS
LIN {X 70.266,Y 97.146,Z 65.719,A 180.000,B 0.000,C 180.000} C_DIS
LIN {X 70.212,Y 96.998,Z 65.714,A 180.000,B 0.000,C 180.000} C_DIS
LIN {X 70.186,Y 96.924,Z 65.711,A 180.000,B 0.000,C 180.000} C_DIS
LIN {X 70.157,Y 96.851,Z 65.708,A 180.000,B 0.000,C 180.000} C_DIS
LIN {X 70.126,Y 96.778,Z 65.706,A 180.000,B 0.000,C 180.000} C_DIS
LIN {X 70.095,Y 96.706,Z 65.703,A 180.000,B 0.000,C 180.000} C_DIS
LIN {X 70.032,Y 96.561,Z 65.697,A 180.000,B 0.000,C 180.000} C_DIS
LIN {X 69.970,Y 96.417,Z 65.692,A 180.000,B 0.000,C 180.000} C_DIS
